HMI tags "2915RS001A01T01"
   "2915RS001A01T01.MSW" : 52809b66-421d-457f-8884-6f7a49d4e247 AT %DB5041.DBX18.0, 500 ms
   "2915RS001A01T01.DefaultText" : TextRef, internal   // Заголовок POPUP окна. При експорте из ECS через скрипт заполняется автоматически, если теги копируются в ручную то требуется в ручную задатать свойство Start Value
   "2915RS001A01T01.BlockInfo" : Array [0..2] of Int AT %DB5041.DBX38.0, 500 ms
   "2915RS001A01T01.StatusWork" : Int AT %DB5041.DBW242, 500 ms
   "2915RS001A01T01.FP_PARAM.DampingTime" : Int AT %DB5041.DBW50, 500 ms
   "2915RS001A01T01.FP_PARAM.Force_Value" : Real AT %DB5041.DBD52, 500 ms
   "2915RS001A01T01.FP_PARAM.Scale_Min" : Real AT %DB5041.DBD56, 500 ms
   "2915RS001A01T01.FP_PARAM.Scale_Max" : Real AT %DB5041.DBD60, 500 ms
   "2915RS001A01T01.FP_PARAM.Gradient" : Real AT %DB5041.DBD64, 500 ms
   "2915RS001A01T01.FP_PARAM.Grad_Pos" : Real AT %DB5041.DBD68, 500 ms
   "2915RS001A01T01.FP_PARAM.Grad_Neg" : Real AT %DB5041.DBD72, 500 ms
   "2915RS001A01T01.FP_PARAM.Grad_X" : Real AT %DB5041.DBD76, 500 ms
   "2915RS001A01T01.FP_PARAM.Gradient_Time_Pre" : Int AT %DB5041.DBW80, 500 ms
   "2915RS001A01T01.FP_PARAM.Gradient_Time_ACC" : Int AT %DB5041.DBW82, 500 ms
   "2915RS001A01T01.FP_PARAM.Alarm_Hyst" : Real AT %DB5041.DBD84, 500 ms
   "2915RS001A01T01.FP_PARAM.AlarmLimit_H3" : Real AT %DB5041.DBD88, 500 ms
   "2915RS001A01T01.FP_PARAM.AlarmLimit_H2" : Real AT %DB5041.DBD92, 500 ms
   "2915RS001A01T01.FP_PARAM.AlarmLimit_H1" : Real AT %DB5041.DBD96, 500 ms
   "2915RS001A01T01.FP_PARAM.AlarmLimit_L1" : Real AT %DB5041.DBD100, 500 ms
   "2915RS001A01T01.FP_PARAM.AlarmLimit_L2" : Real AT %DB5041.DBD104, 500 ms
   "2915RS001A01T01.FP_PARAM.AlarmLimit_L3" : Real AT %DB5041.DBD108, 500 ms
   "2915RS001A01T01.FP_PARAM.AlarmDelay_H3_Pre" : Int AT %DB5041.DBW112, 500 ms
   "2915RS001A01T01.FP_PARAM.AlarmDelay_H3_Acc" : Int AT %DB5041.DBW114, 500 ms
   "2915RS001A01T01.FP_PARAM.AlarmDelay_H2_Pre" : Int AT %DB5041.DBW116, 500 ms
   "2915RS001A01T01.FP_PARAM.AlarmDelay_H2_Acc" : Int AT %DB5041.DBW118, 500 ms
   "2915RS001A01T01.FP_PARAM.AlarmDelay_H1_Pre" : Int AT %DB5041.DBW120, 500 ms
   "2915RS001A01T01.FP_PARAM.AlarmDelay_H1_Acc" : Int AT %DB5041.DBW122, 500 ms
   "2915RS001A01T01.FP_PARAM.AlarmDelay_L1_Pre" : Int AT %DB5041.DBW124, 500 ms
   "2915RS001A01T01.FP_PARAM.AlarmDelay_L1_Acc" : Int AT %DB5041.DBW126, 500 ms
   "2915RS001A01T01.FP_PARAM.AlarmDelay_L2_Pre" : Int AT %DB5041.DBW128, 500 ms
   "2915RS001A01T01.FP_PARAM.AlarmDelay_L2_Acc" : Int AT %DB5041.DBW130, 500 ms
   "2915RS001A01T01.FP_PARAM.AlarmDelay_L3_Pre" : Int AT %DB5041.DBW132, 500 ms
   "2915RS001A01T01.FP_PARAM.AlarmDelay_L3_Acc" : Int AT %DB5041.DBW134, 500 ms
   "2915RS001A01T01.FP_PARAM.OpenLoopDelay_Pre" : Int AT %DB5041.DBW136, 500 ms
   "2915RS001A01T01.FP_PARAM.OpenLoopDelay_Acc" : Int AT %DB5041.DBW138, 500 ms
   "2915RS001A01T01.FP_PARAM.OverRangeDelay_Pre" : Int AT %DB5041.DBW140, 500 ms
   "2915RS001A01T01.FP_PARAM.OverRangeDelay_Acc" : Int AT %DB5041.DBW142, 500 ms
   "2915RS001A01T01.FP_PARAM.AuxLimit_H2_Value" : Real AT %DB5041.DBD144, 500 ms
   "2915RS001A01T01.FP_PARAM.AuxLimit_H1_Value" : Real AT %DB5041.DBD148, 500 ms
   "2915RS001A01T01.FP_PARAM.AuxLimit_L2_Value" : Real AT %DB5041.DBD152, 500 ms
   "2915RS001A01T01.FP_PARAM.AuxLimit_L1_Value" : Real AT %DB5041.DBD156, 500 ms
   "2915RS001A01T01.Unit" : TextRef, internal   // Еденицы измерения При експорте из ECS через скрипт заполняется автоматически, если теги копируются в ручную то требуется задатать свойство Text
   "2915RS001A01T01.Decimals" : TextRef, internal   // Формат отображения При експорте из ECS через скрипт, заполняется автоматически. Если теги копируются в ручную то требуется задатать свойство Text s999999.9
   "2915RS001A01T01.FP_EN.Square" : Bool AT %DB5041.DBX46.0, 500 ms
   "2915RS001A01T01.FP_EN.SquareRoot" : Bool AT %DB5041.DBX46.1, 500 ms
   "2915RS001A01T01.FP_EN.ParentSupress" : Bool AT %DB5041.DBX46.2, 500 ms
   "2915RS001A01T01.FP_EN.ParentSupressUnit" : Bool AT %DB5041.DBX46.3, 500 ms
   "2915RS001A01T01.FP_EN.Force" : Bool AT %DB5041.DBX46.4, 500 ms
   "2915RS001A01T01.FP_EN.Damping" : Bool AT %DB5041.DBX46.5, 500 ms
   "2915RS001A01T01.FP_EN.Gradient_Pos" : Bool AT %DB5041.DBX46.6, 500 ms
   "2915RS001A01T01.FP_EN.Gradient_Neg" : Bool AT %DB5041.DBX46.7, 500 ms
   "2915RS001A01T01.FP_EN.Hysteresis" : Bool AT %DB5041.DBX47.0, 500 ms
   "2915RS001A01T01.FP_EN.Alarm_H3" : Bool AT %DB5041.DBX47.1, 500 ms
   "2915RS001A01T01.FP_EN.Alarm_H2" : Bool AT %DB5041.DBX47.2, 500 ms
   "2915RS001A01T01.FP_EN.Alarm_H1" : Bool AT %DB5041.DBX47.3, 500 ms
   "2915RS001A01T01.FP_EN.Alarm_L1" : Bool AT %DB5041.DBX47.4, 500 ms
   "2915RS001A01T01.FP_EN.Alarm_L2" : Bool AT %DB5041.DBX47.5, 500 ms
   "2915RS001A01T01.FP_EN.Alarm_L3" : Bool AT %DB5041.DBX47.6, 500 ms
   "2915RS001A01T01.FP_EN.AlarmDelay_H3" : Bool AT %DB5041.DBX47.7, 500 ms
   "2915RS001A01T01.FP_EN.AlarmDelay_H2" : Bool AT %DB5041.DBX48.0, 500 ms
   "2915RS001A01T01.FP_EN.AlarmDelay_H1" : Bool AT %DB5041.DBX48.1, 500 ms
   "2915RS001A01T01.FP_EN.AlarmDelay_L1" : Bool AT %DB5041.DBX48.2, 500 ms
   "2915RS001A01T01.FP_EN.AlarmDelay_L2" : Bool AT %DB5041.DBX48.3, 500 ms
   "2915RS001A01T01.FP_EN.AlarmDelay_L3" : Bool AT %DB5041.DBX48.4, 500 ms
   "2915RS001A01T01.FP_EN.ROC_Warn" : Bool AT %DB5041.DBX48.5, 500 ms
   "2915RS001A01T01.FP_EN.U_Range_Warn" : Bool AT %DB5041.DBX48.6, 500 ms
   "2915RS001A01T01.FP_EN.O_Range_Warn" : Bool AT %DB5041.DBX48.7, 500 ms
   "2915RS001A01T01.trend_tag_name" : TextRef, internal   // Еденицы измерения При експорте из ECS через скрипт - заполняется автоматически, если теги копируются в ручную то требуется задатать свойство Text - имя тега для тренда
   "2915RS001A01T01.DQ.AL_H3" : Bool AT %DB5041.DBX16.0, 500 ms
   "2915RS001A01T01.DQ.AL_H2" : Bool AT %DB5041.DBX16.1, 500 ms
   "2915RS001A01T01.DQ.AL_H1" : Bool AT %DB5041.DBX16.2, 500 ms
   "2915RS001A01T01.DQ.AL_L1" : Bool AT %DB5041.DBX16.3, 500 ms
   "2915RS001A01T01.DQ.AL_L2" : Bool AT %DB5041.DBX16.4, 500 ms
   "2915RS001A01T01.DQ.AL_L3" : Bool AT %DB5041.DBX16.5, 500 ms
   "2915RS001A01T01.DQ.SIG_OK" : Bool AT %DB5041.DBX16.6, 500 ms
   "2915RS001A01T01.DQ.LIM_H2" : Bool AT %DB5041.DBX16.7, 500 ms
   "2915RS001A01T01.DQ.LIM_H1" : Bool AT %DB5041.DBX17.0, 500 ms
   "2915RS001A01T01.DQ.LIM_L1" : Bool AT %DB5041.DBX17.1, 500 ms
   "2915RS001A01T01.DQ.LIM_L2" : Bool AT %DB5041.DBX17.2, 500 ms
   "2915RS001A01T01.DQ.GR_P" : Bool AT %DB5041.DBX17.3, 500 ms
   "2915RS001A01T01.DQ.GR_N" : Bool AT %DB5041.DBX17.4, 500 ms
   "2915RS001A01T01.I.IN" : Real AT %DB5041.DBD2, 500 ms
   "2915RS001A01T01.I.SIG_TYPE" : Int AT %DB5041.DBW0, 500 ms
   "2915RS001A01T01.I.FI_BUS" : Byte AT %DB5041.DBB6, 500 ms
   "2915RS001A01T01.DI.U_RANGE" : Bool AT %DB5041.DBX7.0, 500 ms
   "2915RS001A01T01.DI.O_RANGE" : Bool AT %DB5041.DBX7.1, 500 ms
   "2915RS001A01T01.DI.SIG_FAULT" : Bool AT %DB5041.DBX7.2, 500 ms
   "2915RS001A01T01.DI.EnConfig" : Bool AT %DB5041.DBX7.3, 500 ms
   "2915RS001A01T01.DI.AEN" : Bool AT %DB5041.DBX7.4, 500 ms
   "2915RS001A01T01.DI.AL_SUPR" : Bool AT %DB5041.DBX7.5, 500 ms
   "2915RS001A01T01.Q.PV_NORM" : Real AT %DB5041.DBD8, 500 ms
   "2915RS001A01T01.Q.PV_SCAL" : Real AT %DB5041.DBD12, 500 ms
   "2915RS001A01T01.ParentInfo" : TextRef, internal   // Имя родителя для попап окна, вкладка инфо. При експорте из ECS через скрипт заполняется автоматически, если теги копируются в ручную то требуется в ручную задатать свойство Start Value

HMI tags "2915RS001A01T02"
   "2915RS001A01T02.MSW" : 52809b66-421d-457f-8884-6f7a49d4e247 AT %DB5042.DBX18.0, 500 ms
   "2915RS001A01T02.DefaultText" : TextRef, internal   // Заголовок POPUP окна. При експорте из ECS через скрипт заполняется автоматически, если теги копируются в ручную то требуется в ручную задатать свойство Start Value
   "2915RS001A01T02.BlockInfo" : Array [0..2] of Int AT %DB5042.DBX38.0, 500 ms
   "2915RS001A01T02.StatusWork" : Int AT %DB5042.DBW242, 500 ms
   "2915RS001A01T02.FP_PARAM.DampingTime" : Int AT %DB5042.DBW50, 500 ms
   "2915RS001A01T02.FP_PARAM.Force_Value" : Real AT %DB5042.DBD52, 500 ms
   "2915RS001A01T02.FP_PARAM.Scale_Min" : Real AT %DB5042.DBD56, 500 ms
   "2915RS001A01T02.FP_PARAM.Scale_Max" : Real AT %DB5042.DBD60, 500 ms
   "2915RS001A01T02.FP_PARAM.Gradient" : Real AT %DB5042.DBD64, 500 ms
   "2915RS001A01T02.FP_PARAM.Grad_Pos" : Real AT %DB5042.DBD68, 500 ms
   "2915RS001A01T02.FP_PARAM.Grad_Neg" : Real AT %DB5042.DBD72, 500 ms
   "2915RS001A01T02.FP_PARAM.Grad_X" : Real AT %DB5042.DBD76, 500 ms
   "2915RS001A01T02.FP_PARAM.Gradient_Time_Pre" : Int AT %DB5042.DBW80, 500 ms
   "2915RS001A01T02.FP_PARAM.Gradient_Time_ACC" : Int AT %DB5042.DBW82, 500 ms
   "2915RS001A01T02.FP_PARAM.Alarm_Hyst" : Real AT %DB5042.DBD84, 500 ms
   "2915RS001A01T02.FP_PARAM.AlarmLimit_H3" : Real AT %DB5042.DBD88, 500 ms
   "2915RS001A01T02.FP_PARAM.AlarmLimit_H2" : Real AT %DB5042.DBD92, 500 ms
   "2915RS001A01T02.FP_PARAM.AlarmLimit_H1" : Real AT %DB5042.DBD96, 500 ms
   "2915RS001A01T02.FP_PARAM.AlarmLimit_L1" : Real AT %DB5042.DBD100, 500 ms
   "2915RS001A01T02.FP_PARAM.AlarmLimit_L2" : Real AT %DB5042.DBD104, 500 ms
   "2915RS001A01T02.FP_PARAM.AlarmLimit_L3" : Real AT %DB5042.DBD108, 500 ms
   "2915RS001A01T02.FP_PARAM.AlarmDelay_H3_Pre" : Int AT %DB5042.DBW112, 500 ms
   "2915RS001A01T02.FP_PARAM.AlarmDelay_H3_Acc" : Int AT %DB5042.DBW114, 500 ms
   "2915RS001A01T02.FP_PARAM.AlarmDelay_H2_Pre" : Int AT %DB5042.DBW116, 500 ms
   "2915RS001A01T02.FP_PARAM.AlarmDelay_H2_Acc" : Int AT %DB5042.DBW118, 500 ms
   "2915RS001A01T02.FP_PARAM.AlarmDelay_H1_Pre" : Int AT %DB5042.DBW120, 500 ms
   "2915RS001A01T02.FP_PARAM.AlarmDelay_H1_Acc" : Int AT %DB5042.DBW122, 500 ms
   "2915RS001A01T02.FP_PARAM.AlarmDelay_L1_Pre" : Int AT %DB5042.DBW124, 500 ms
   "2915RS001A01T02.FP_PARAM.AlarmDelay_L1_Acc" : Int AT %DB5042.DBW126, 500 ms
   "2915RS001A01T02.FP_PARAM.AlarmDelay_L2_Pre" : Int AT %DB5042.DBW128, 500 ms
   "2915RS001A01T02.FP_PARAM.AlarmDelay_L2_Acc" : Int AT %DB5042.DBW130, 500 ms
   "2915RS001A01T02.FP_PARAM.AlarmDelay_L3_Pre" : Int AT %DB5042.DBW132, 500 ms
   "2915RS001A01T02.FP_PARAM.AlarmDelay_L3_Acc" : Int AT %DB5042.DBW134, 500 ms
   "2915RS001A01T02.FP_PARAM.OpenLoopDelay_Pre" : Int AT %DB5042.DBW136, 500 ms
   "2915RS001A01T02.FP_PARAM.OpenLoopDelay_Acc" : Int AT %DB5042.DBW138, 500 ms
   "2915RS001A01T02.FP_PARAM.OverRangeDelay_Pre" : Int AT %DB5042.DBW140, 500 ms
   "2915RS001A01T02.FP_PARAM.OverRangeDelay_Acc" : Int AT %DB5042.DBW142, 500 ms
   "2915RS001A01T02.FP_PARAM.AuxLimit_H2_Value" : Real AT %DB5042.DBD144, 500 ms
   "2915RS001A01T02.FP_PARAM.AuxLimit_H1_Value" : Real AT %DB5042.DBD148, 500 ms
   "2915RS001A01T02.FP_PARAM.AuxLimit_L2_Value" : Real AT %DB5042.DBD152, 500 ms
   "2915RS001A01T02.FP_PARAM.AuxLimit_L1_Value" : Real AT %DB5042.DBD156, 500 ms
   "2915RS001A01T02.Unit" : TextRef, internal   // Еденицы измерения При експорте из ECS через скрипт заполняется автоматически, если теги копируются в ручную то требуется задатать свойство Text
   "2915RS001A01T02.Decimals" : TextRef, internal   // Формат отображения При експорте из ECS через скрипт, заполняется автоматически. Если теги копируются в ручную то требуется задатать свойство Text s999999.9
   "2915RS001A01T02.FP_EN.Square" : Bool AT %DB5042.DBX46.0, 500 ms
   "2915RS001A01T02.FP_EN.SquareRoot" : Bool AT %DB5042.DBX46.1, 500 ms
   "2915RS001A01T02.FP_EN.ParentSupress" : Bool AT %DB5042.DBX46.2, 500 ms
   "2915RS001A01T02.FP_EN.ParentSupressUnit" : Bool AT %DB5042.DBX46.3, 500 ms
   "2915RS001A01T02.FP_EN.Force" : Bool AT %DB5042.DBX46.4, 500 ms
   "2915RS001A01T02.FP_EN.Damping" : Bool AT %DB5042.DBX46.5, 500 ms
   "2915RS001A01T02.FP_EN.Gradient_Pos" : Bool AT %DB5042.DBX46.6, 500 ms
   "2915RS001A01T02.FP_EN.Gradient_Neg" : Bool AT %DB5042.DBX46.7, 500 ms
   "2915RS001A01T02.FP_EN.Hysteresis" : Bool AT %DB5042.DBX47.0, 500 ms
   "2915RS001A01T02.FP_EN.Alarm_H3" : Bool AT %DB5042.DBX47.1, 500 ms
   "2915RS001A01T02.FP_EN.Alarm_H2" : Bool AT %DB5042.DBX47.2, 500 ms
   "2915RS001A01T02.FP_EN.Alarm_H1" : Bool AT %DB5042.DBX47.3, 500 ms
   "2915RS001A01T02.FP_EN.Alarm_L1" : Bool AT %DB5042.DBX47.4, 500 ms
   "2915RS001A01T02.FP_EN.Alarm_L2" : Bool AT %DB5042.DBX47.5, 500 ms
   "2915RS001A01T02.FP_EN.Alarm_L3" : Bool AT %DB5042.DBX47.6, 500 ms
   "2915RS001A01T02.FP_EN.AlarmDelay_H3" : Bool AT %DB5042.DBX47.7, 500 ms
   "2915RS001A01T02.FP_EN.AlarmDelay_H2" : Bool AT %DB5042.DBX48.0, 500 ms
   "2915RS001A01T02.FP_EN.AlarmDelay_H1" : Bool AT %DB5042.DBX48.1, 500 ms
   "2915RS001A01T02.FP_EN.AlarmDelay_L1" : Bool AT %DB5042.DBX48.2, 500 ms
   "2915RS001A01T02.FP_EN.AlarmDelay_L2" : Bool AT %DB5042.DBX48.3, 500 ms
   "2915RS001A01T02.FP_EN.AlarmDelay_L3" : Bool AT %DB5042.DBX48.4, 500 ms
   "2915RS001A01T02.FP_EN.ROC_Warn" : Bool AT %DB5042.DBX48.5, 500 ms
   "2915RS001A01T02.FP_EN.U_Range_Warn" : Bool AT %DB5042.DBX48.6, 500 ms
   "2915RS001A01T02.FP_EN.O_Range_Warn" : Bool AT %DB5042.DBX48.7, 500 ms
   "2915RS001A01T02.trend_tag_name" : TextRef, internal   // Еденицы измерения При експорте из ECS через скрипт - заполняется автоматически, если теги копируются в ручную то требуется задатать свойство Text - имя тега для тренда
   "2915RS001A01T02.DQ.AL_H3" : Bool AT %DB5042.DBX16.0, 500 ms
   "2915RS001A01T02.DQ.AL_H2" : Bool AT %DB5042.DBX16.1, 500 ms
   "2915RS001A01T02.DQ.AL_H1" : Bool AT %DB5042.DBX16.2, 500 ms
   "2915RS001A01T02.DQ.AL_L1" : Bool AT %DB5042.DBX16.3, 500 ms
   "2915RS001A01T02.DQ.AL_L2" : Bool AT %DB5042.DBX16.4, 500 ms
   "2915RS001A01T02.DQ.AL_L3" : Bool AT %DB5042.DBX16.5, 500 ms
   "2915RS001A01T02.DQ.SIG_OK" : Bool AT %DB5042.DBX16.6, 500 ms
   "2915RS001A01T02.DQ.LIM_H2" : Bool AT %DB5042.DBX16.7, 500 ms
   "2915RS001A01T02.DQ.LIM_H1" : Bool AT %DB5042.DBX17.0, 500 ms
   "2915RS001A01T02.DQ.LIM_L1" : Bool AT %DB5042.DBX17.1, 500 ms
   "2915RS001A01T02.DQ.LIM_L2" : Bool AT %DB5042.DBX17.2, 500 ms
   "2915RS001A01T02.DQ.GR_P" : Bool AT %DB5042.DBX17.3, 500 ms
   "2915RS001A01T02.DQ.GR_N" : Bool AT %DB5042.DBX17.4, 500 ms
   "2915RS001A01T02.I.IN" : Real AT %DB5042.DBD2, 500 ms
   "2915RS001A01T02.I.SIG_TYPE" : Int AT %DB5042.DBW0, 500 ms
   "2915RS001A01T02.I.FI_BUS" : Byte AT %DB5042.DBB6, 500 ms
   "2915RS001A01T02.DI.U_RANGE" : Bool AT %DB5042.DBX7.0, 500 ms
   "2915RS001A01T02.DI.O_RANGE" : Bool AT %DB5042.DBX7.1, 500 ms
   "2915RS001A01T02.DI.SIG_FAULT" : Bool AT %DB5042.DBX7.2, 500 ms
   "2915RS001A01T02.DI.EnConfig" : Bool AT %DB5042.DBX7.3, 500 ms
   "2915RS001A01T02.DI.AEN" : Bool AT %DB5042.DBX7.4, 500 ms
   "2915RS001A01T02.DI.AL_SUPR" : Bool AT %DB5042.DBX7.5, 500 ms
   "2915RS001A01T02.Q.PV_NORM" : Real AT %DB5042.DBD8, 500 ms
   "2915RS001A01T02.Q.PV_SCAL" : Real AT %DB5042.DBD12, 500 ms
   "2915RS001A01T02.ParentInfo" : TextRef, internal   // Имя родителя для попап окна, вкладка инфо. При експорте из ECS через скрипт заполняется автоматически, если теги копируются в ручную то требуется в ручную задатать свойство Start Value

HMI tags "2915RS001A01T03"
   "2915RS001A01T03.MSW" : 52809b66-421d-457f-8884-6f7a49d4e247 AT %DB5043.DBX18.0, 500 ms
   "2915RS001A01T03.DefaultText" : TextRef, internal   // Заголовок POPUP окна. При експорте из ECS через скрипт заполняется автоматически, если теги копируются в ручную то требуется в ручную задатать свойство Start Value
   "2915RS001A01T03.BlockInfo" : Array [0..2] of Int AT %DB5043.DBX38.0, 500 ms
   "2915RS001A01T03.StatusWork" : Int AT %DB5043.DBW242, 500 ms
   "2915RS001A01T03.FP_PARAM.DampingTime" : Int AT %DB5043.DBW50, 500 ms
   "2915RS001A01T03.FP_PARAM.Force_Value" : Real AT %DB5043.DBD52, 500 ms
   "2915RS001A01T03.FP_PARAM.Scale_Min" : Real AT %DB5043.DBD56, 500 ms
   "2915RS001A01T03.FP_PARAM.Scale_Max" : Real AT %DB5043.DBD60, 500 ms
   "2915RS001A01T03.FP_PARAM.Gradient" : Real AT %DB5043.DBD64, 500 ms
   "2915RS001A01T03.FP_PARAM.Grad_Pos" : Real AT %DB5043.DBD68, 500 ms
   "2915RS001A01T03.FP_PARAM.Grad_Neg" : Real AT %DB5043.DBD72, 500 ms
   "2915RS001A01T03.FP_PARAM.Grad_X" : Real AT %DB5043.DBD76, 500 ms
   "2915RS001A01T03.FP_PARAM.Gradient_Time_Pre" : Int AT %DB5043.DBW80, 500 ms
   "2915RS001A01T03.FP_PARAM.Gradient_Time_ACC" : Int AT %DB5043.DBW82, 500 ms
   "2915RS001A01T03.FP_PARAM.Alarm_Hyst" : Real AT %DB5043.DBD84, 500 ms
   "2915RS001A01T03.FP_PARAM.AlarmLimit_H3" : Real AT %DB5043.DBD88, 500 ms
   "2915RS001A01T03.FP_PARAM.AlarmLimit_H2" : Real AT %DB5043.DBD92, 500 ms
   "2915RS001A01T03.FP_PARAM.AlarmLimit_H1" : Real AT %DB5043.DBD96, 500 ms
   "2915RS001A01T03.FP_PARAM.AlarmLimit_L1" : Real AT %DB5043.DBD100, 500 ms
   "2915RS001A01T03.FP_PARAM.AlarmLimit_L2" : Real AT %DB5043.DBD104, 500 ms
   "2915RS001A01T03.FP_PARAM.AlarmLimit_L3" : Real AT %DB5043.DBD108, 500 ms
   "2915RS001A01T03.FP_PARAM.AlarmDelay_H3_Pre" : Int AT %DB5043.DBW112, 500 ms
   "2915RS001A01T03.FP_PARAM.AlarmDelay_H3_Acc" : Int AT %DB5043.DBW114, 500 ms
   "2915RS001A01T03.FP_PARAM.AlarmDelay_H2_Pre" : Int AT %DB5043.DBW116, 500 ms
   "2915RS001A01T03.FP_PARAM.AlarmDelay_H2_Acc" : Int AT %DB5043.DBW118, 500 ms
   "2915RS001A01T03.FP_PARAM.AlarmDelay_H1_Pre" : Int AT %DB5043.DBW120, 500 ms
   "2915RS001A01T03.FP_PARAM.AlarmDelay_H1_Acc" : Int AT %DB5043.DBW122, 500 ms
   "2915RS001A01T03.FP_PARAM.AlarmDelay_L1_Pre" : Int AT %DB5043.DBW124, 500 ms
   "2915RS001A01T03.FP_PARAM.AlarmDelay_L1_Acc" : Int AT %DB5043.DBW126, 500 ms
   "2915RS001A01T03.FP_PARAM.AlarmDelay_L2_Pre" : Int AT %DB5043.DBW128, 500 ms
   "2915RS001A01T03.FP_PARAM.AlarmDelay_L2_Acc" : Int AT %DB5043.DBW130, 500 ms
   "2915RS001A01T03.FP_PARAM.AlarmDelay_L3_Pre" : Int AT %DB5043.DBW132, 500 ms
   "2915RS001A01T03.FP_PARAM.AlarmDelay_L3_Acc" : Int AT %DB5043.DBW134, 500 ms
   "2915RS001A01T03.FP_PARAM.OpenLoopDelay_Pre" : Int AT %DB5043.DBW136, 500 ms
   "2915RS001A01T03.FP_PARAM.OpenLoopDelay_Acc" : Int AT %DB5043.DBW138, 500 ms
   "2915RS001A01T03.FP_PARAM.OverRangeDelay_Pre" : Int AT %DB5043.DBW140, 500 ms
   "2915RS001A01T03.FP_PARAM.OverRangeDelay_Acc" : Int AT %DB5043.DBW142, 500 ms
   "2915RS001A01T03.FP_PARAM.AuxLimit_H2_Value" : Real AT %DB5043.DBD144, 500 ms
   "2915RS001A01T03.FP_PARAM.AuxLimit_H1_Value" : Real AT %DB5043.DBD148, 500 ms
   "2915RS001A01T03.FP_PARAM.AuxLimit_L2_Value" : Real AT %DB5043.DBD152, 500 ms
   "2915RS001A01T03.FP_PARAM.AuxLimit_L1_Value" : Real AT %DB5043.DBD156, 500 ms
   "2915RS001A01T03.Unit" : TextRef, internal   // Еденицы измерения При експорте из ECS через скрипт заполняется автоматически, если теги копируются в ручную то требуется задатать свойство Text
   "2915RS001A01T03.Decimals" : TextRef, internal   // Формат отображения При експорте из ECS через скрипт, заполняется автоматически. Если теги копируются в ручную то требуется задатать свойство Text s999999.9
   "2915RS001A01T03.FP_EN.Square" : Bool AT %DB5043.DBX46.0, 500 ms
   "2915RS001A01T03.FP_EN.SquareRoot" : Bool AT %DB5043.DBX46.1, 500 ms
   "2915RS001A01T03.FP_EN.ParentSupress" : Bool AT %DB5043.DBX46.2, 500 ms
   "2915RS001A01T03.FP_EN.ParentSupressUnit" : Bool AT %DB5043.DBX46.3, 500 ms
   "2915RS001A01T03.FP_EN.Force" : Bool AT %DB5043.DBX46.4, 500 ms
   "2915RS001A01T03.FP_EN.Damping" : Bool AT %DB5043.DBX46.5, 500 ms
   "2915RS001A01T03.FP_EN.Gradient_Pos" : Bool AT %DB5043.DBX46.6, 500 ms
   "2915RS001A01T03.FP_EN.Gradient_Neg" : Bool AT %DB5043.DBX46.7, 500 ms
   "2915RS001A01T03.FP_EN.Hysteresis" : Bool AT %DB5043.DBX47.0, 500 ms
   "2915RS001A01T03.FP_EN.Alarm_H3" : Bool AT %DB5043.DBX47.1, 500 ms
   "2915RS001A01T03.FP_EN.Alarm_H2" : Bool AT %DB5043.DBX47.2, 500 ms
   "2915RS001A01T03.FP_EN.Alarm_H1" : Bool AT %DB5043.DBX47.3, 500 ms
   "2915RS001A01T03.FP_EN.Alarm_L1" : Bool AT %DB5043.DBX47.4, 500 ms
   "2915RS001A01T03.FP_EN.Alarm_L2" : Bool AT %DB5043.DBX47.5, 500 ms
   "2915RS001A01T03.FP_EN.Alarm_L3" : Bool AT %DB5043.DBX47.6, 500 ms
   "2915RS001A01T03.FP_EN.AlarmDelay_H3" : Bool AT %DB5043.DBX47.7, 500 ms
   "2915RS001A01T03.FP_EN.AlarmDelay_H2" : Bool AT %DB5043.DBX48.0, 500 ms
   "2915RS001A01T03.FP_EN.AlarmDelay_H1" : Bool AT %DB5043.DBX48.1, 500 ms
   "2915RS001A01T03.FP_EN.AlarmDelay_L1" : Bool AT %DB5043.DBX48.2, 500 ms
   "2915RS001A01T03.FP_EN.AlarmDelay_L2" : Bool AT %DB5043.DBX48.3, 500 ms
   "2915RS001A01T03.FP_EN.AlarmDelay_L3" : Bool AT %DB5043.DBX48.4, 500 ms
   "2915RS001A01T03.FP_EN.ROC_Warn" : Bool AT %DB5043.DBX48.5, 500 ms
   "2915RS001A01T03.FP_EN.U_Range_Warn" : Bool AT %DB5043.DBX48.6, 500 ms
   "2915RS001A01T03.FP_EN.O_Range_Warn" : Bool AT %DB5043.DBX48.7, 500 ms
   "2915RS001A01T03.trend_tag_name" : TextRef, internal   // Еденицы измерения При експорте из ECS через скрипт - заполняется автоматически, если теги копируются в ручную то требуется задатать свойство Text - имя тега для тренда
   "2915RS001A01T03.DQ.AL_H3" : Bool AT %DB5043.DBX16.0, 500 ms
   "2915RS001A01T03.DQ.AL_H2" : Bool AT %DB5043.DBX16.1, 500 ms
   "2915RS001A01T03.DQ.AL_H1" : Bool AT %DB5043.DBX16.2, 500 ms
   "2915RS001A01T03.DQ.AL_L1" : Bool AT %DB5043.DBX16.3, 500 ms
   "2915RS001A01T03.DQ.AL_L2" : Bool AT %DB5043.DBX16.4, 500 ms
   "2915RS001A01T03.DQ.AL_L3" : Bool AT %DB5043.DBX16.5, 500 ms
   "2915RS001A01T03.DQ.SIG_OK" : Bool AT %DB5043.DBX16.6, 500 ms
   "2915RS001A01T03.DQ.LIM_H2" : Bool AT %DB5043.DBX16.7, 500 ms
   "2915RS001A01T03.DQ.LIM_H1" : Bool AT %DB5043.DBX17.0, 500 ms
   "2915RS001A01T03.DQ.LIM_L1" : Bool AT %DB5043.DBX17.1, 500 ms
   "2915RS001A01T03.DQ.LIM_L2" : Bool AT %DB5043.DBX17.2, 500 ms
   "2915RS001A01T03.DQ.GR_P" : Bool AT %DB5043.DBX17.3, 500 ms
   "2915RS001A01T03.DQ.GR_N" : Bool AT %DB5043.DBX17.4, 500 ms
   "2915RS001A01T03.I.IN" : Real AT %DB5043.DBD2, 500 ms
   "2915RS001A01T03.I.SIG_TYPE" : Int AT %DB5043.DBW0, 500 ms
   "2915RS001A01T03.I.FI_BUS" : Byte AT %DB5043.DBB6, 500 ms
   "2915RS001A01T03.DI.U_RANGE" : Bool AT %DB5043.DBX7.0, 500 ms
   "2915RS001A01T03.DI.O_RANGE" : Bool AT %DB5043.DBX7.1, 500 ms
   "2915RS001A01T03.DI.SIG_FAULT" : Bool AT %DB5043.DBX7.2, 500 ms
   "2915RS001A01T03.DI.EnConfig" : Bool AT %DB5043.DBX7.3, 500 ms
   "2915RS001A01T03.DI.AEN" : Bool AT %DB5043.DBX7.4, 500 ms
   "2915RS001A01T03.DI.AL_SUPR" : Bool AT %DB5043.DBX7.5, 500 ms
   "2915RS001A01T03.Q.PV_NORM" : Real AT %DB5043.DBD8, 500 ms
   "2915RS001A01T03.Q.PV_SCAL" : Real AT %DB5043.DBD12, 500 ms
   "2915RS001A01T03.ParentInfo" : TextRef, internal   // Имя родителя для попап окна, вкладка инфо. При експорте из ECS через скрипт заполняется автоматически, если теги копируются в ручную то требуется в ручную задатать свойство Start Value

HMI tags "2915RS001A01T04"
   "2915RS001A01T04.MSW" : 52809b66-421d-457f-8884-6f7a49d4e247 AT %DB5044.DBX18.0, 500 ms
   "2915RS001A01T04.DefaultText" : TextRef, internal   // Заголовок POPUP окна. При експорте из ECS через скрипт заполняется автоматически, если теги копируются в ручную то требуется в ручную задатать свойство Start Value
   "2915RS001A01T04.BlockInfo" : Array [0..2] of Int AT %DB5044.DBX38.0, 500 ms
   "2915RS001A01T04.StatusWork" : Int AT %DB5044.DBW242, 500 ms
   "2915RS001A01T04.FP_PARAM.DampingTime" : Int AT %DB5044.DBW50, 500 ms
   "2915RS001A01T04.FP_PARAM.Force_Value" : Real AT %DB5044.DBD52, 500 ms
   "2915RS001A01T04.FP_PARAM.Scale_Min" : Real AT %DB5044.DBD56, 500 ms
   "2915RS001A01T04.FP_PARAM.Scale_Max" : Real AT %DB5044.DBD60, 500 ms
   "2915RS001A01T04.FP_PARAM.Gradient" : Real AT %DB5044.DBD64, 500 ms
   "2915RS001A01T04.FP_PARAM.Grad_Pos" : Real AT %DB5044.DBD68, 500 ms
   "2915RS001A01T04.FP_PARAM.Grad_Neg" : Real AT %DB5044.DBD72, 500 ms
   "2915RS001A01T04.FP_PARAM.Grad_X" : Real AT %DB5044.DBD76, 500 ms
   "2915RS001A01T04.FP_PARAM.Gradient_Time_Pre" : Int AT %DB5044.DBW80, 500 ms
   "2915RS001A01T04.FP_PARAM.Gradient_Time_ACC" : Int AT %DB5044.DBW82, 500 ms
   "2915RS001A01T04.FP_PARAM.Alarm_Hyst" : Real AT %DB5044.DBD84, 500 ms
   "2915RS001A01T04.FP_PARAM.AlarmLimit_H3" : Real AT %DB5044.DBD88, 500 ms
   "2915RS001A01T04.FP_PARAM.AlarmLimit_H2" : Real AT %DB5044.DBD92, 500 ms
   "2915RS001A01T04.FP_PARAM.AlarmLimit_H1" : Real AT %DB5044.DBD96, 500 ms
   "2915RS001A01T04.FP_PARAM.AlarmLimit_L1" : Real AT %DB5044.DBD100, 500 ms
   "2915RS001A01T04.FP_PARAM.AlarmLimit_L2" : Real AT %DB5044.DBD104, 500 ms
   "2915RS001A01T04.FP_PARAM.AlarmLimit_L3" : Real AT %DB5044.DBD108, 500 ms
   "2915RS001A01T04.FP_PARAM.AlarmDelay_H3_Pre" : Int AT %DB5044.DBW112, 500 ms
   "2915RS001A01T04.FP_PARAM.AlarmDelay_H3_Acc" : Int AT %DB5044.DBW114, 500 ms
   "2915RS001A01T04.FP_PARAM.AlarmDelay_H2_Pre" : Int AT %DB5044.DBW116, 500 ms
   "2915RS001A01T04.FP_PARAM.AlarmDelay_H2_Acc" : Int AT %DB5044.DBW118, 500 ms
   "2915RS001A01T04.FP_PARAM.AlarmDelay_H1_Pre" : Int AT %DB5044.DBW120, 500 ms
   "2915RS001A01T04.FP_PARAM.AlarmDelay_H1_Acc" : Int AT %DB5044.DBW122, 500 ms
   "2915RS001A01T04.FP_PARAM.AlarmDelay_L1_Pre" : Int AT %DB5044.DBW124, 500 ms
   "2915RS001A01T04.FP_PARAM.AlarmDelay_L1_Acc" : Int AT %DB5044.DBW126, 500 ms
   "2915RS001A01T04.FP_PARAM.AlarmDelay_L2_Pre" : Int AT %DB5044.DBW128, 500 ms
   "2915RS001A01T04.FP_PARAM.AlarmDelay_L2_Acc" : Int AT %DB5044.DBW130, 500 ms
   "2915RS001A01T04.FP_PARAM.AlarmDelay_L3_Pre" : Int AT %DB5044.DBW132, 500 ms
   "2915RS001A01T04.FP_PARAM.AlarmDelay_L3_Acc" : Int AT %DB5044.DBW134, 500 ms
   "2915RS001A01T04.FP_PARAM.OpenLoopDelay_Pre" : Int AT %DB5044.DBW136, 500 ms
   "2915RS001A01T04.FP_PARAM.OpenLoopDelay_Acc" : Int AT %DB5044.DBW138, 500 ms
   "2915RS001A01T04.FP_PARAM.OverRangeDelay_Pre" : Int AT %DB5044.DBW140, 500 ms
   "2915RS001A01T04.FP_PARAM.OverRangeDelay_Acc" : Int AT %DB5044.DBW142, 500 ms
   "2915RS001A01T04.FP_PARAM.AuxLimit_H2_Value" : Real AT %DB5044.DBD144, 500 ms
   "2915RS001A01T04.FP_PARAM.AuxLimit_H1_Value" : Real AT %DB5044.DBD148, 500 ms
   "2915RS001A01T04.FP_PARAM.AuxLimit_L2_Value" : Real AT %DB5044.DBD152, 500 ms
   "2915RS001A01T04.FP_PARAM.AuxLimit_L1_Value" : Real AT %DB5044.DBD156, 500 ms
   "2915RS001A01T04.Unit" : TextRef, internal   // Еденицы измерения При експорте из ECS через скрипт заполняется автоматически, если теги копируются в ручную то требуется задатать свойство Text
   "2915RS001A01T04.Decimals" : TextRef, internal   // Формат отображения При експорте из ECS через скрипт, заполняется автоматически. Если теги копируются в ручную то требуется задатать свойство Text s999999.9
   "2915RS001A01T04.FP_EN.Square" : Bool AT %DB5044.DBX46.0, 500 ms
   "2915RS001A01T04.FP_EN.SquareRoot" : Bool AT %DB5044.DBX46.1, 500 ms
   "2915RS001A01T04.FP_EN.ParentSupress" : Bool AT %DB5044.DBX46.2, 500 ms
   "2915RS001A01T04.FP_EN.ParentSupressUnit" : Bool AT %DB5044.DBX46.3, 500 ms
   "2915RS001A01T04.FP_EN.Force" : Bool AT %DB5044.DBX46.4, 500 ms
   "2915RS001A01T04.FP_EN.Damping" : Bool AT %DB5044.DBX46.5, 500 ms
   "2915RS001A01T04.FP_EN.Gradient_Pos" : Bool AT %DB5044.DBX46.6, 500 ms
   "2915RS001A01T04.FP_EN.Gradient_Neg" : Bool AT %DB5044.DBX46.7, 500 ms
   "2915RS001A01T04.FP_EN.Hysteresis" : Bool AT %DB5044.DBX47.0, 500 ms
   "2915RS001A01T04.FP_EN.Alarm_H3" : Bool AT %DB5044.DBX47.1, 500 ms
   "2915RS001A01T04.FP_EN.Alarm_H2" : Bool AT %DB5044.DBX47.2, 500 ms
   "2915RS001A01T04.FP_EN.Alarm_H1" : Bool AT %DB5044.DBX47.3, 500 ms
   "2915RS001A01T04.FP_EN.Alarm_L1" : Bool AT %DB5044.DBX47.4, 500 ms
   "2915RS001A01T04.FP_EN.Alarm_L2" : Bool AT %DB5044.DBX47.5, 500 ms
   "2915RS001A01T04.FP_EN.Alarm_L3" : Bool AT %DB5044.DBX47.6, 500 ms
   "2915RS001A01T04.FP_EN.AlarmDelay_H3" : Bool AT %DB5044.DBX47.7, 500 ms
   "2915RS001A01T04.FP_EN.AlarmDelay_H2" : Bool AT %DB5044.DBX48.0, 500 ms
   "2915RS001A01T04.FP_EN.AlarmDelay_H1" : Bool AT %DB5044.DBX48.1, 500 ms
   "2915RS001A01T04.FP_EN.AlarmDelay_L1" : Bool AT %DB5044.DBX48.2, 500 ms
   "2915RS001A01T04.FP_EN.AlarmDelay_L2" : Bool AT %DB5044.DBX48.3, 500 ms
   "2915RS001A01T04.FP_EN.AlarmDelay_L3" : Bool AT %DB5044.DBX48.4, 500 ms
   "2915RS001A01T04.FP_EN.ROC_Warn" : Bool AT %DB5044.DBX48.5, 500 ms
   "2915RS001A01T04.FP_EN.U_Range_Warn" : Bool AT %DB5044.DBX48.6, 500 ms
   "2915RS001A01T04.FP_EN.O_Range_Warn" : Bool AT %DB5044.DBX48.7, 500 ms
   "2915RS001A01T04.trend_tag_name" : TextRef, internal   // Еденицы измерения При експорте из ECS через скрипт - заполняется автоматически, если теги копируются в ручную то требуется задатать свойство Text - имя тега для тренда
   "2915RS001A01T04.DQ.AL_H3" : Bool AT %DB5044.DBX16.0, 500 ms
   "2915RS001A01T04.DQ.AL_H2" : Bool AT %DB5044.DBX16.1, 500 ms
   "2915RS001A01T04.DQ.AL_H1" : Bool AT %DB5044.DBX16.2, 500 ms
   "2915RS001A01T04.DQ.AL_L1" : Bool AT %DB5044.DBX16.3, 500 ms
   "2915RS001A01T04.DQ.AL_L2" : Bool AT %DB5044.DBX16.4, 500 ms
   "2915RS001A01T04.DQ.AL_L3" : Bool AT %DB5044.DBX16.5, 500 ms
   "2915RS001A01T04.DQ.SIG_OK" : Bool AT %DB5044.DBX16.6, 500 ms
   "2915RS001A01T04.DQ.LIM_H2" : Bool AT %DB5044.DBX16.7, 500 ms
   "2915RS001A01T04.DQ.LIM_H1" : Bool AT %DB5044.DBX17.0, 500 ms
   "2915RS001A01T04.DQ.LIM_L1" : Bool AT %DB5044.DBX17.1, 500 ms
   "2915RS001A01T04.DQ.LIM_L2" : Bool AT %DB5044.DBX17.2, 500 ms
   "2915RS001A01T04.DQ.GR_P" : Bool AT %DB5044.DBX17.3, 500 ms
   "2915RS001A01T04.DQ.GR_N" : Bool AT %DB5044.DBX17.4, 500 ms
   "2915RS001A01T04.I.IN" : Real AT %DB5044.DBD2, 500 ms
   "2915RS001A01T04.I.SIG_TYPE" : Int AT %DB5044.DBW0, 500 ms
   "2915RS001A01T04.I.FI_BUS" : Byte AT %DB5044.DBB6, 500 ms
   "2915RS001A01T04.DI.U_RANGE" : Bool AT %DB5044.DBX7.0, 500 ms
   "2915RS001A01T04.DI.O_RANGE" : Bool AT %DB5044.DBX7.1, 500 ms
   "2915RS001A01T04.DI.SIG_FAULT" : Bool AT %DB5044.DBX7.2, 500 ms
   "2915RS001A01T04.DI.EnConfig" : Bool AT %DB5044.DBX7.3, 500 ms
   "2915RS001A01T04.DI.AEN" : Bool AT %DB5044.DBX7.4, 500 ms
   "2915RS001A01T04.DI.AL_SUPR" : Bool AT %DB5044.DBX7.5, 500 ms
   "2915RS001A01T04.Q.PV_NORM" : Real AT %DB5044.DBD8, 500 ms
   "2915RS001A01T04.Q.PV_SCAL" : Real AT %DB5044.DBD12, 500 ms
   "2915RS001A01T04.ParentInfo" : TextRef, internal   // Имя родителя для попап окна, вкладка инфо. При експорте из ECS через скрипт заполняется автоматически, если теги копируются в ручную то требуется в ручную задатать свойство Start Value

HMI tags "2915RS001A01T05"
   "2915RS001A01T05.MSW" : 52809b66-421d-457f-8884-6f7a49d4e247 AT %DB5045.DBX18.0, 500 ms
   "2915RS001A01T05.DefaultText" : TextRef, internal   // Заголовок POPUP окна. При експорте из ECS через скрипт заполняется автоматически, если теги копируются в ручную то требуется в ручную задатать свойство Start Value
   "2915RS001A01T05.BlockInfo" : Array [0..2] of Int AT %DB5045.DBX38.0, 500 ms
   "2915RS001A01T05.StatusWork" : Int AT %DB5045.DBW242, 500 ms
   "2915RS001A01T05.FP_PARAM.DampingTime" : Int AT %DB5045.DBW50, 500 ms
   "2915RS001A01T05.FP_PARAM.Force_Value" : Real AT %DB5045.DBD52, 500 ms
   "2915RS001A01T05.FP_PARAM.Scale_Min" : Real AT %DB5045.DBD56, 500 ms
   "2915RS001A01T05.FP_PARAM.Scale_Max" : Real AT %DB5045.DBD60, 500 ms
   "2915RS001A01T05.FP_PARAM.Gradient" : Real AT %DB5045.DBD64, 500 ms
   "2915RS001A01T05.FP_PARAM.Grad_Pos" : Real AT %DB5045.DBD68, 500 ms
   "2915RS001A01T05.FP_PARAM.Grad_Neg" : Real AT %DB5045.DBD72, 500 ms
   "2915RS001A01T05.FP_PARAM.Grad_X" : Real AT %DB5045.DBD76, 500 ms
   "2915RS001A01T05.FP_PARAM.Gradient_Time_Pre" : Int AT %DB5045.DBW80, 500 ms
   "2915RS001A01T05.FP_PARAM.Gradient_Time_ACC" : Int AT %DB5045.DBW82, 500 ms
   "2915RS001A01T05.FP_PARAM.Alarm_Hyst" : Real AT %DB5045.DBD84, 500 ms
   "2915RS001A01T05.FP_PARAM.AlarmLimit_H3" : Real AT %DB5045.DBD88, 500 ms
   "2915RS001A01T05.FP_PARAM.AlarmLimit_H2" : Real AT %DB5045.DBD92, 500 ms
   "2915RS001A01T05.FP_PARAM.AlarmLimit_H1" : Real AT %DB5045.DBD96, 500 ms
   "2915RS001A01T05.FP_PARAM.AlarmLimit_L1" : Real AT %DB5045.DBD100, 500 ms
   "2915RS001A01T05.FP_PARAM.AlarmLimit_L2" : Real AT %DB5045.DBD104, 500 ms
   "2915RS001A01T05.FP_PARAM.AlarmLimit_L3" : Real AT %DB5045.DBD108, 500 ms
   "2915RS001A01T05.FP_PARAM.AlarmDelay_H3_Pre" : Int AT %DB5045.DBW112, 500 ms
   "2915RS001A01T05.FP_PARAM.AlarmDelay_H3_Acc" : Int AT %DB5045.DBW114, 500 ms
   "2915RS001A01T05.FP_PARAM.AlarmDelay_H2_Pre" : Int AT %DB5045.DBW116, 500 ms
   "2915RS001A01T05.FP_PARAM.AlarmDelay_H2_Acc" : Int AT %DB5045.DBW118, 500 ms
   "2915RS001A01T05.FP_PARAM.AlarmDelay_H1_Pre" : Int AT %DB5045.DBW120, 500 ms
   "2915RS001A01T05.FP_PARAM.AlarmDelay_H1_Acc" : Int AT %DB5045.DBW122, 500 ms
   "2915RS001A01T05.FP_PARAM.AlarmDelay_L1_Pre" : Int AT %DB5045.DBW124, 500 ms
   "2915RS001A01T05.FP_PARAM.AlarmDelay_L1_Acc" : Int AT %DB5045.DBW126, 500 ms
   "2915RS001A01T05.FP_PARAM.AlarmDelay_L2_Pre" : Int AT %DB5045.DBW128, 500 ms
   "2915RS001A01T05.FP_PARAM.AlarmDelay_L2_Acc" : Int AT %DB5045.DBW130, 500 ms
   "2915RS001A01T05.FP_PARAM.AlarmDelay_L3_Pre" : Int AT %DB5045.DBW132, 500 ms
   "2915RS001A01T05.FP_PARAM.AlarmDelay_L3_Acc" : Int AT %DB5045.DBW134, 500 ms
   "2915RS001A01T05.FP_PARAM.OpenLoopDelay_Pre" : Int AT %DB5045.DBW136, 500 ms
   "2915RS001A01T05.FP_PARAM.OpenLoopDelay_Acc" : Int AT %DB5045.DBW138, 500 ms
   "2915RS001A01T05.FP_PARAM.OverRangeDelay_Pre" : Int AT %DB5045.DBW140, 500 ms
   "2915RS001A01T05.FP_PARAM.OverRangeDelay_Acc" : Int AT %DB5045.DBW142, 500 ms
   "2915RS001A01T05.FP_PARAM.AuxLimit_H2_Value" : Real AT %DB5045.DBD144, 500 ms
   "2915RS001A01T05.FP_PARAM.AuxLimit_H1_Value" : Real AT %DB5045.DBD148, 500 ms
   "2915RS001A01T05.FP_PARAM.AuxLimit_L2_Value" : Real AT %DB5045.DBD152, 500 ms
   "2915RS001A01T05.FP_PARAM.AuxLimit_L1_Value" : Real AT %DB5045.DBD156, 500 ms
   "2915RS001A01T05.Unit" : TextRef, internal   // Еденицы измерения При експорте из ECS через скрипт заполняется автоматически, если теги копируются в ручную то требуется задатать свойство Text
   "2915RS001A01T05.Decimals" : TextRef, internal   // Формат отображения При експорте из ECS через скрипт, заполняется автоматически. Если теги копируются в ручную то требуется задатать свойство Text s999999.9
   "2915RS001A01T05.FP_EN.Square" : Bool AT %DB5045.DBX46.0, 500 ms
   "2915RS001A01T05.FP_EN.SquareRoot" : Bool AT %DB5045.DBX46.1, 500 ms
   "2915RS001A01T05.FP_EN.ParentSupress" : Bool AT %DB5045.DBX46.2, 500 ms
   "2915RS001A01T05.FP_EN.ParentSupressUnit" : Bool AT %DB5045.DBX46.3, 500 ms
   "2915RS001A01T05.FP_EN.Force" : Bool AT %DB5045.DBX46.4, 500 ms
   "2915RS001A01T05.FP_EN.Damping" : Bool AT %DB5045.DBX46.5, 500 ms
   "2915RS001A01T05.FP_EN.Gradient_Pos" : Bool AT %DB5045.DBX46.6, 500 ms
   "2915RS001A01T05.FP_EN.Gradient_Neg" : Bool AT %DB5045.DBX46.7, 500 ms
   "2915RS001A01T05.FP_EN.Hysteresis" : Bool AT %DB5045.DBX47.0, 500 ms
   "2915RS001A01T05.FP_EN.Alarm_H3" : Bool AT %DB5045.DBX47.1, 500 ms
   "2915RS001A01T05.FP_EN.Alarm_H2" : Bool AT %DB5045.DBX47.2, 500 ms
   "2915RS001A01T05.FP_EN.Alarm_H1" : Bool AT %DB5045.DBX47.3, 500 ms
   "2915RS001A01T05.FP_EN.Alarm_L1" : Bool AT %DB5045.DBX47.4, 500 ms
   "2915RS001A01T05.FP_EN.Alarm_L2" : Bool AT %DB5045.DBX47.5, 500 ms
   "2915RS001A01T05.FP_EN.Alarm_L3" : Bool AT %DB5045.DBX47.6, 500 ms
   "2915RS001A01T05.FP_EN.AlarmDelay_H3" : Bool AT %DB5045.DBX47.7, 500 ms
   "2915RS001A01T05.FP_EN.AlarmDelay_H2" : Bool AT %DB5045.DBX48.0, 500 ms
   "2915RS001A01T05.FP_EN.AlarmDelay_H1" : Bool AT %DB5045.DBX48.1, 500 ms
   "2915RS001A01T05.FP_EN.AlarmDelay_L1" : Bool AT %DB5045.DBX48.2, 500 ms
   "2915RS001A01T05.FP_EN.AlarmDelay_L2" : Bool AT %DB5045.DBX48.3, 500 ms
   "2915RS001A01T05.FP_EN.AlarmDelay_L3" : Bool AT %DB5045.DBX48.4, 500 ms
   "2915RS001A01T05.FP_EN.ROC_Warn" : Bool AT %DB5045.DBX48.5, 500 ms
   "2915RS001A01T05.FP_EN.U_Range_Warn" : Bool AT %DB5045.DBX48.6, 500 ms
   "2915RS001A01T05.FP_EN.O_Range_Warn" : Bool AT %DB5045.DBX48.7, 500 ms
   "2915RS001A01T05.trend_tag_name" : TextRef, internal   // Еденицы измерения При експорте из ECS через скрипт - заполняется автоматически, если теги копируются в ручную то требуется задатать свойство Text - имя тега для тренда
   "2915RS001A01T05.DQ.AL_H3" : Bool AT %DB5045.DBX16.0, 500 ms
   "2915RS001A01T05.DQ.AL_H2" : Bool AT %DB5045.DBX16.1, 500 ms
   "2915RS001A01T05.DQ.AL_H1" : Bool AT %DB5045.DBX16.2, 500 ms
   "2915RS001A01T05.DQ.AL_L1" : Bool AT %DB5045.DBX16.3, 500 ms
   "2915RS001A01T05.DQ.AL_L2" : Bool AT %DB5045.DBX16.4, 500 ms
   "2915RS001A01T05.DQ.AL_L3" : Bool AT %DB5045.DBX16.5, 500 ms
   "2915RS001A01T05.DQ.SIG_OK" : Bool AT %DB5045.DBX16.6, 500 ms
   "2915RS001A01T05.DQ.LIM_H2" : Bool AT %DB5045.DBX16.7, 500 ms
   "2915RS001A01T05.DQ.LIM_H1" : Bool AT %DB5045.DBX17.0, 500 ms
   "2915RS001A01T05.DQ.LIM_L1" : Bool AT %DB5045.DBX17.1, 500 ms
   "2915RS001A01T05.DQ.LIM_L2" : Bool AT %DB5045.DBX17.2, 500 ms
   "2915RS001A01T05.DQ.GR_P" : Bool AT %DB5045.DBX17.3, 500 ms
   "2915RS001A01T05.DQ.GR_N" : Bool AT %DB5045.DBX17.4, 500 ms
   "2915RS001A01T05.I.IN" : Real AT %DB5045.DBD2, 500 ms
   "2915RS001A01T05.I.SIG_TYPE" : Int AT %DB5045.DBW0, 500 ms
   "2915RS001A01T05.I.FI_BUS" : Byte AT %DB5045.DBB6, 500 ms
   "2915RS001A01T05.DI.U_RANGE" : Bool AT %DB5045.DBX7.0, 500 ms
   "2915RS001A01T05.DI.O_RANGE" : Bool AT %DB5045.DBX7.1, 500 ms
   "2915RS001A01T05.DI.SIG_FAULT" : Bool AT %DB5045.DBX7.2, 500 ms
   "2915RS001A01T05.DI.EnConfig" : Bool AT %DB5045.DBX7.3, 500 ms
   "2915RS001A01T05.DI.AEN" : Bool AT %DB5045.DBX7.4, 500 ms
   "2915RS001A01T05.DI.AL_SUPR" : Bool AT %DB5045.DBX7.5, 500 ms
   "2915RS001A01T05.Q.PV_NORM" : Real AT %DB5045.DBD8, 500 ms
   "2915RS001A01T05.Q.PV_SCAL" : Real AT %DB5045.DBD12, 500 ms
   "2915RS001A01T05.ParentInfo" : TextRef, internal   // Имя родителя для попап окна, вкладка инфо. При експорте из ECS через скрипт заполняется автоматически, если теги копируются в ручную то требуется в ручную задатать свойство Start Value

HMI tags "2915RS001N01T01"
   "2915RS001N01T01.MSW" : 52809b66-421d-457f-8884-6f7a49d4e247 AT %DB5303.DBX18.0, 500 ms
   "2915RS001N01T01.DefaultText" : TextRef, internal   // Заголовок POPUP окна. При експорте из ECS через скрипт заполняется автоматически, если теги копируются в ручную то требуется в ручную задатать свойство Start Value
   "2915RS001N01T01.BlockInfo" : Array [0..2] of Int AT %DB5303.DBX38.0, 500 ms
   "2915RS001N01T01.StatusWork" : Int AT %DB5303.DBW242, 500 ms
   "2915RS001N01T01.FP_PARAM.DampingTime" : Int AT %DB5303.DBW50, 500 ms
   "2915RS001N01T01.FP_PARAM.Force_Value" : Real AT %DB5303.DBD52, 500 ms
   "2915RS001N01T01.FP_PARAM.Scale_Min" : Real AT %DB5303.DBD56, 500 ms
   "2915RS001N01T01.FP_PARAM.Scale_Max" : Real AT %DB5303.DBD60, 500 ms
   "2915RS001N01T01.FP_PARAM.Gradient" : Real AT %DB5303.DBD64, 500 ms
   "2915RS001N01T01.FP_PARAM.Grad_Pos" : Real AT %DB5303.DBD68, 500 ms
   "2915RS001N01T01.FP_PARAM.Grad_Neg" : Real AT %DB5303.DBD72, 500 ms
   "2915RS001N01T01.FP_PARAM.Grad_X" : Real AT %DB5303.DBD76, 500 ms
   "2915RS001N01T01.FP_PARAM.Gradient_Time_Pre" : Int AT %DB5303.DBW80, 500 ms
   "2915RS001N01T01.FP_PARAM.Gradient_Time_ACC" : Int AT %DB5303.DBW82, 500 ms
   "2915RS001N01T01.FP_PARAM.Alarm_Hyst" : Real AT %DB5303.DBD84, 500 ms
   "2915RS001N01T01.FP_PARAM.AlarmLimit_H3" : Real AT %DB5303.DBD88, 500 ms
   "2915RS001N01T01.FP_PARAM.AlarmLimit_H2" : Real AT %DB5303.DBD92, 500 ms
   "2915RS001N01T01.FP_PARAM.AlarmLimit_H1" : Real AT %DB5303.DBD96, 500 ms
   "2915RS001N01T01.FP_PARAM.AlarmLimit_L1" : Real AT %DB5303.DBD100, 500 ms
   "2915RS001N01T01.FP_PARAM.AlarmLimit_L2" : Real AT %DB5303.DBD104, 500 ms
   "2915RS001N01T01.FP_PARAM.AlarmLimit_L3" : Real AT %DB5303.DBD108, 500 ms
   "2915RS001N01T01.FP_PARAM.AlarmDelay_H3_Pre" : Int AT %DB5303.DBW112, 500 ms
   "2915RS001N01T01.FP_PARAM.AlarmDelay_H3_Acc" : Int AT %DB5303.DBW114, 500 ms
   "2915RS001N01T01.FP_PARAM.AlarmDelay_H2_Pre" : Int AT %DB5303.DBW116, 500 ms
   "2915RS001N01T01.FP_PARAM.AlarmDelay_H2_Acc" : Int AT %DB5303.DBW118, 500 ms
   "2915RS001N01T01.FP_PARAM.AlarmDelay_H1_Pre" : Int AT %DB5303.DBW120, 500 ms
   "2915RS001N01T01.FP_PARAM.AlarmDelay_H1_Acc" : Int AT %DB5303.DBW122, 500 ms
   "2915RS001N01T01.FP_PARAM.AlarmDelay_L1_Pre" : Int AT %DB5303.DBW124, 500 ms
   "2915RS001N01T01.FP_PARAM.AlarmDelay_L1_Acc" : Int AT %DB5303.DBW126, 500 ms
   "2915RS001N01T01.FP_PARAM.AlarmDelay_L2_Pre" : Int AT %DB5303.DBW128, 500 ms
   "2915RS001N01T01.FP_PARAM.AlarmDelay_L2_Acc" : Int AT %DB5303.DBW130, 500 ms
   "2915RS001N01T01.FP_PARAM.AlarmDelay_L3_Pre" : Int AT %DB5303.DBW132, 500 ms
   "2915RS001N01T01.FP_PARAM.AlarmDelay_L3_Acc" : Int AT %DB5303.DBW134, 500 ms
   "2915RS001N01T01.FP_PARAM.OpenLoopDelay_Pre" : Int AT %DB5303.DBW136, 500 ms
   "2915RS001N01T01.FP_PARAM.OpenLoopDelay_Acc" : Int AT %DB5303.DBW138, 500 ms
   "2915RS001N01T01.FP_PARAM.OverRangeDelay_Pre" : Int AT %DB5303.DBW140, 500 ms
   "2915RS001N01T01.FP_PARAM.OverRangeDelay_Acc" : Int AT %DB5303.DBW142, 500 ms
   "2915RS001N01T01.FP_PARAM.AuxLimit_H2_Value" : Real AT %DB5303.DBD144, 500 ms
   "2915RS001N01T01.FP_PARAM.AuxLimit_H1_Value" : Real AT %DB5303.DBD148, 500 ms
   "2915RS001N01T01.FP_PARAM.AuxLimit_L2_Value" : Real AT %DB5303.DBD152, 500 ms
   "2915RS001N01T01.FP_PARAM.AuxLimit_L1_Value" : Real AT %DB5303.DBD156, 500 ms
   "2915RS001N01T01.Unit" : TextRef, internal   // Еденицы измерения При експорте из ECS через скрипт заполняется автоматически, если теги копируются в ручную то требуется задатать свойство Text
   "2915RS001N01T01.Decimals" : TextRef, internal   // Формат отображения При експорте из ECS через скрипт, заполняется автоматически. Если теги копируются в ручную то требуется задатать свойство Text s999999.9
   "2915RS001N01T01.FP_EN.Square" : Bool AT %DB5303.DBX46.0, 500 ms
   "2915RS001N01T01.FP_EN.SquareRoot" : Bool AT %DB5303.DBX46.1, 500 ms
   "2915RS001N01T01.FP_EN.ParentSupress" : Bool AT %DB5303.DBX46.2, 500 ms
   "2915RS001N01T01.FP_EN.ParentSupressUnit" : Bool AT %DB5303.DBX46.3, 500 ms
   "2915RS001N01T01.FP_EN.Force" : Bool AT %DB5303.DBX46.4, 500 ms
   "2915RS001N01T01.FP_EN.Damping" : Bool AT %DB5303.DBX46.5, 500 ms
   "2915RS001N01T01.FP_EN.Gradient_Pos" : Bool AT %DB5303.DBX46.6, 500 ms
   "2915RS001N01T01.FP_EN.Gradient_Neg" : Bool AT %DB5303.DBX46.7, 500 ms
   "2915RS001N01T01.FP_EN.Hysteresis" : Bool AT %DB5303.DBX47.0, 500 ms
   "2915RS001N01T01.FP_EN.Alarm_H3" : Bool AT %DB5303.DBX47.1, 500 ms
   "2915RS001N01T01.FP_EN.Alarm_H2" : Bool AT %DB5303.DBX47.2, 500 ms
   "2915RS001N01T01.FP_EN.Alarm_H1" : Bool AT %DB5303.DBX47.3, 500 ms
   "2915RS001N01T01.FP_EN.Alarm_L1" : Bool AT %DB5303.DBX47.4, 500 ms
   "2915RS001N01T01.FP_EN.Alarm_L2" : Bool AT %DB5303.DBX47.5, 500 ms
   "2915RS001N01T01.FP_EN.Alarm_L3" : Bool AT %DB5303.DBX47.6, 500 ms
   "2915RS001N01T01.FP_EN.AlarmDelay_H3" : Bool AT %DB5303.DBX47.7, 500 ms
   "2915RS001N01T01.FP_EN.AlarmDelay_H2" : Bool AT %DB5303.DBX48.0, 500 ms
   "2915RS001N01T01.FP_EN.AlarmDelay_H1" : Bool AT %DB5303.DBX48.1, 500 ms
   "2915RS001N01T01.FP_EN.AlarmDelay_L1" : Bool AT %DB5303.DBX48.2, 500 ms
   "2915RS001N01T01.FP_EN.AlarmDelay_L2" : Bool AT %DB5303.DBX48.3, 500 ms
   "2915RS001N01T01.FP_EN.AlarmDelay_L3" : Bool AT %DB5303.DBX48.4, 500 ms
   "2915RS001N01T01.FP_EN.ROC_Warn" : Bool AT %DB5303.DBX48.5, 500 ms
   "2915RS001N01T01.FP_EN.U_Range_Warn" : Bool AT %DB5303.DBX48.6, 500 ms
   "2915RS001N01T01.FP_EN.O_Range_Warn" : Bool AT %DB5303.DBX48.7, 500 ms
   "2915RS001N01T01.trend_tag_name" : TextRef, internal   // Еденицы измерения При експорте из ECS через скрипт - заполняется автоматически, если теги копируются в ручную то требуется задатать свойство Text - имя тега для тренда
   "2915RS001N01T01.DQ.AL_H3" : Bool AT %DB5303.DBX16.0, 500 ms
   "2915RS001N01T01.DQ.AL_H2" : Bool AT %DB5303.DBX16.1, 500 ms
   "2915RS001N01T01.DQ.AL_H1" : Bool AT %DB5303.DBX16.2, 500 ms
   "2915RS001N01T01.DQ.AL_L1" : Bool AT %DB5303.DBX16.3, 500 ms
   "2915RS001N01T01.DQ.AL_L2" : Bool AT %DB5303.DBX16.4, 500 ms
   "2915RS001N01T01.DQ.AL_L3" : Bool AT %DB5303.DBX16.5, 500 ms
   "2915RS001N01T01.DQ.SIG_OK" : Bool AT %DB5303.DBX16.6, 500 ms
   "2915RS001N01T01.DQ.LIM_H2" : Bool AT %DB5303.DBX16.7, 500 ms
   "2915RS001N01T01.DQ.LIM_H1" : Bool AT %DB5303.DBX17.0, 500 ms
   "2915RS001N01T01.DQ.LIM_L1" : Bool AT %DB5303.DBX17.1, 500 ms
   "2915RS001N01T01.DQ.LIM_L2" : Bool AT %DB5303.DBX17.2, 500 ms
   "2915RS001N01T01.DQ.GR_P" : Bool AT %DB5303.DBX17.3, 500 ms
   "2915RS001N01T01.DQ.GR_N" : Bool AT %DB5303.DBX17.4, 500 ms
   "2915RS001N01T01.I.IN" : Real AT %DB5303.DBD2, 500 ms
   "2915RS001N01T01.I.SIG_TYPE" : Int AT %DB5303.DBW0, 500 ms
   "2915RS001N01T01.I.FI_BUS" : Byte AT %DB5303.DBB6, 500 ms
   "2915RS001N01T01.DI.U_RANGE" : Bool AT %DB5303.DBX7.0, 500 ms
   "2915RS001N01T01.DI.O_RANGE" : Bool AT %DB5303.DBX7.1, 500 ms
   "2915RS001N01T01.DI.SIG_FAULT" : Bool AT %DB5303.DBX7.2, 500 ms
   "2915RS001N01T01.DI.EnConfig" : Bool AT %DB5303.DBX7.3, 500 ms
   "2915RS001N01T01.DI.AEN" : Bool AT %DB5303.DBX7.4, 500 ms
   "2915RS001N01T01.DI.AL_SUPR" : Bool AT %DB5303.DBX7.5, 500 ms
   "2915RS001N01T01.Q.PV_NORM" : Real AT %DB5303.DBD8, 500 ms
   "2915RS001N01T01.Q.PV_SCAL" : Real AT %DB5303.DBD12, 500 ms
   "2915RS001N01T01.ParentInfo" : TextRef, internal   // Имя родителя для попап окна, вкладка инфо. При експорте из ECS через скрипт заполняется автоматически, если теги копируются в ручную то требуется в ручную задатать свойство Start Value

HMI tags "2920RS001A01A01"
   "2920RS001A01A01.MSW" : 52809b66-421d-457f-8884-6f7a49d4e247 AT %DB5046.DBX18.0, 500 ms
   "2920RS001A01A01.DefaultText" : TextRef, internal   // Заголовок POPUP окна. При експорте из ECS через скрипт заполняется автоматически, если теги копируются в ручную то требуется в ручную задатать свойство Start Value
   "2920RS001A01A01.BlockInfo" : Array [0..2] of Int AT %DB5046.DBX38.0, 500 ms
   "2920RS001A01A01.StatusWork" : Int AT %DB5046.DBW242, 500 ms
   "2920RS001A01A01.FP_PARAM.DampingTime" : Int AT %DB5046.DBW50, 500 ms
   "2920RS001A01A01.FP_PARAM.Force_Value" : Real AT %DB5046.DBD52, 500 ms
   "2920RS001A01A01.FP_PARAM.Scale_Min" : Real AT %DB5046.DBD56, 500 ms
   "2920RS001A01A01.FP_PARAM.Scale_Max" : Real AT %DB5046.DBD60, 500 ms
   "2920RS001A01A01.FP_PARAM.Gradient" : Real AT %DB5046.DBD64, 500 ms
   "2920RS001A01A01.FP_PARAM.Grad_Pos" : Real AT %DB5046.DBD68, 500 ms
   "2920RS001A01A01.FP_PARAM.Grad_Neg" : Real AT %DB5046.DBD72, 500 ms
   "2920RS001A01A01.FP_PARAM.Grad_X" : Real AT %DB5046.DBD76, 500 ms
   "2920RS001A01A01.FP_PARAM.Gradient_Time_Pre" : Int AT %DB5046.DBW80, 500 ms
   "2920RS001A01A01.FP_PARAM.Gradient_Time_ACC" : Int AT %DB5046.DBW82, 500 ms
   "2920RS001A01A01.FP_PARAM.Alarm_Hyst" : Real AT %DB5046.DBD84, 500 ms
   "2920RS001A01A01.FP_PARAM.AlarmLimit_H3" : Real AT %DB5046.DBD88, 500 ms
   "2920RS001A01A01.FP_PARAM.AlarmLimit_H2" : Real AT %DB5046.DBD92, 500 ms
   "2920RS001A01A01.FP_PARAM.AlarmLimit_H1" : Real AT %DB5046.DBD96, 500 ms
   "2920RS001A01A01.FP_PARAM.AlarmLimit_L1" : Real AT %DB5046.DBD100, 500 ms
   "2920RS001A01A01.FP_PARAM.AlarmLimit_L2" : Real AT %DB5046.DBD104, 500 ms
   "2920RS001A01A01.FP_PARAM.AlarmLimit_L3" : Real AT %DB5046.DBD108, 500 ms
   "2920RS001A01A01.FP_PARAM.AlarmDelay_H3_Pre" : Int AT %DB5046.DBW112, 500 ms
   "2920RS001A01A01.FP_PARAM.AlarmDelay_H3_Acc" : Int AT %DB5046.DBW114, 500 ms
   "2920RS001A01A01.FP_PARAM.AlarmDelay_H2_Pre" : Int AT %DB5046.DBW116, 500 ms
   "2920RS001A01A01.FP_PARAM.AlarmDelay_H2_Acc" : Int AT %DB5046.DBW118, 500 ms
   "2920RS001A01A01.FP_PARAM.AlarmDelay_H1_Pre" : Int AT %DB5046.DBW120, 500 ms
   "2920RS001A01A01.FP_PARAM.AlarmDelay_H1_Acc" : Int AT %DB5046.DBW122, 500 ms
   "2920RS001A01A01.FP_PARAM.AlarmDelay_L1_Pre" : Int AT %DB5046.DBW124, 500 ms
   "2920RS001A01A01.FP_PARAM.AlarmDelay_L1_Acc" : Int AT %DB5046.DBW126, 500 ms
   "2920RS001A01A01.FP_PARAM.AlarmDelay_L2_Pre" : Int AT %DB5046.DBW128, 500 ms
   "2920RS001A01A01.FP_PARAM.AlarmDelay_L2_Acc" : Int AT %DB5046.DBW130, 500 ms
   "2920RS001A01A01.FP_PARAM.AlarmDelay_L3_Pre" : Int AT %DB5046.DBW132, 500 ms
   "2920RS001A01A01.FP_PARAM.AlarmDelay_L3_Acc" : Int AT %DB5046.DBW134, 500 ms
   "2920RS001A01A01.FP_PARAM.OpenLoopDelay_Pre" : Int AT %DB5046.DBW136, 500 ms
   "2920RS001A01A01.FP_PARAM.OpenLoopDelay_Acc" : Int AT %DB5046.DBW138, 500 ms
   "2920RS001A01A01.FP_PARAM.OverRangeDelay_Pre" : Int AT %DB5046.DBW140, 500 ms
   "2920RS001A01A01.FP_PARAM.OverRangeDelay_Acc" : Int AT %DB5046.DBW142, 500 ms
   "2920RS001A01A01.FP_PARAM.AuxLimit_H2_Value" : Real AT %DB5046.DBD144, 500 ms
   "2920RS001A01A01.FP_PARAM.AuxLimit_H1_Value" : Real AT %DB5046.DBD148, 500 ms
   "2920RS001A01A01.FP_PARAM.AuxLimit_L2_Value" : Real AT %DB5046.DBD152, 500 ms
   "2920RS001A01A01.FP_PARAM.AuxLimit_L1_Value" : Real AT %DB5046.DBD156, 500 ms
   "2920RS001A01A01.Unit" : TextRef, internal   // Еденицы измерения При експорте из ECS через скрипт заполняется автоматически, если теги копируются в ручную то требуется задатать свойство Text
   "2920RS001A01A01.Decimals" : TextRef, internal   // Формат отображения При експорте из ECS через скрипт, заполняется автоматически. Если теги копируются в ручную то требуется задатать свойство Text s999999.9
   "2920RS001A01A01.FP_EN.Square" : Bool AT %DB5046.DBX46.0, 500 ms
   "2920RS001A01A01.FP_EN.SquareRoot" : Bool AT %DB5046.DBX46.1, 500 ms
   "2920RS001A01A01.FP_EN.ParentSupress" : Bool AT %DB5046.DBX46.2, 500 ms
   "2920RS001A01A01.FP_EN.ParentSupressUnit" : Bool AT %DB5046.DBX46.3, 500 ms
   "2920RS001A01A01.FP_EN.Force" : Bool AT %DB5046.DBX46.4, 500 ms
   "2920RS001A01A01.FP_EN.Damping" : Bool AT %DB5046.DBX46.5, 500 ms
   "2920RS001A01A01.FP_EN.Gradient_Pos" : Bool AT %DB5046.DBX46.6, 500 ms
   "2920RS001A01A01.FP_EN.Gradient_Neg" : Bool AT %DB5046.DBX46.7, 500 ms
   "2920RS001A01A01.FP_EN.Hysteresis" : Bool AT %DB5046.DBX47.0, 500 ms
   "2920RS001A01A01.FP_EN.Alarm_H3" : Bool AT %DB5046.DBX47.1, 500 ms
   "2920RS001A01A01.FP_EN.Alarm_H2" : Bool AT %DB5046.DBX47.2, 500 ms
   "2920RS001A01A01.FP_EN.Alarm_H1" : Bool AT %DB5046.DBX47.3, 500 ms
   "2920RS001A01A01.FP_EN.Alarm_L1" : Bool AT %DB5046.DBX47.4, 500 ms
   "2920RS001A01A01.FP_EN.Alarm_L2" : Bool AT %DB5046.DBX47.5, 500 ms
   "2920RS001A01A01.FP_EN.Alarm_L3" : Bool AT %DB5046.DBX47.6, 500 ms
   "2920RS001A01A01.FP_EN.AlarmDelay_H3" : Bool AT %DB5046.DBX47.7, 500 ms
   "2920RS001A01A01.FP_EN.AlarmDelay_H2" : Bool AT %DB5046.DBX48.0, 500 ms
   "2920RS001A01A01.FP_EN.AlarmDelay_H1" : Bool AT %DB5046.DBX48.1, 500 ms
   "2920RS001A01A01.FP_EN.AlarmDelay_L1" : Bool AT %DB5046.DBX48.2, 500 ms
   "2920RS001A01A01.FP_EN.AlarmDelay_L2" : Bool AT %DB5046.DBX48.3, 500 ms
   "2920RS001A01A01.FP_EN.AlarmDelay_L3" : Bool AT %DB5046.DBX48.4, 500 ms
   "2920RS001A01A01.FP_EN.ROC_Warn" : Bool AT %DB5046.DBX48.5, 500 ms
   "2920RS001A01A01.FP_EN.U_Range_Warn" : Bool AT %DB5046.DBX48.6, 500 ms
   "2920RS001A01A01.FP_EN.O_Range_Warn" : Bool AT %DB5046.DBX48.7, 500 ms
   "2920RS001A01A01.trend_tag_name" : TextRef, internal   // Еденицы измерения При експорте из ECS через скрипт - заполняется автоматически, если теги копируются в ручную то требуется задатать свойство Text - имя тега для тренда
   "2920RS001A01A01.DQ.AL_H3" : Bool AT %DB5046.DBX16.0, 500 ms
   "2920RS001A01A01.DQ.AL_H2" : Bool AT %DB5046.DBX16.1, 500 ms
   "2920RS001A01A01.DQ.AL_H1" : Bool AT %DB5046.DBX16.2, 500 ms
   "2920RS001A01A01.DQ.AL_L1" : Bool AT %DB5046.DBX16.3, 500 ms
   "2920RS001A01A01.DQ.AL_L2" : Bool AT %DB5046.DBX16.4, 500 ms
   "2920RS001A01A01.DQ.AL_L3" : Bool AT %DB5046.DBX16.5, 500 ms
   "2920RS001A01A01.DQ.SIG_OK" : Bool AT %DB5046.DBX16.6, 500 ms
   "2920RS001A01A01.DQ.LIM_H2" : Bool AT %DB5046.DBX16.7, 500 ms
   "2920RS001A01A01.DQ.LIM_H1" : Bool AT %DB5046.DBX17.0, 500 ms
   "2920RS001A01A01.DQ.LIM_L1" : Bool AT %DB5046.DBX17.1, 500 ms
   "2920RS001A01A01.DQ.LIM_L2" : Bool AT %DB5046.DBX17.2, 500 ms
   "2920RS001A01A01.DQ.GR_P" : Bool AT %DB5046.DBX17.3, 500 ms
   "2920RS001A01A01.DQ.GR_N" : Bool AT %DB5046.DBX17.4, 500 ms
   "2920RS001A01A01.I.IN" : Real AT %DB5046.DBD2, 500 ms
   "2920RS001A01A01.I.SIG_TYPE" : Int AT %DB5046.DBW0, 500 ms
   "2920RS001A01A01.I.FI_BUS" : Byte AT %DB5046.DBB6, 500 ms
   "2920RS001A01A01.DI.U_RANGE" : Bool AT %DB5046.DBX7.0, 500 ms
   "2920RS001A01A01.DI.O_RANGE" : Bool AT %DB5046.DBX7.1, 500 ms
   "2920RS001A01A01.DI.SIG_FAULT" : Bool AT %DB5046.DBX7.2, 500 ms
   "2920RS001A01A01.DI.EnConfig" : Bool AT %DB5046.DBX7.3, 500 ms
   "2920RS001A01A01.DI.AEN" : Bool AT %DB5046.DBX7.4, 500 ms
   "2920RS001A01A01.DI.AL_SUPR" : Bool AT %DB5046.DBX7.5, 500 ms
   "2920RS001A01A01.Q.PV_NORM" : Real AT %DB5046.DBD8, 500 ms
   "2920RS001A01A01.Q.PV_SCAL" : Real AT %DB5046.DBD12, 500 ms
   "2920RS001A01A01.ParentInfo" : TextRef, internal   // Имя родителя для попап окна, вкладка инфо. При експорте из ECS через скрипт заполняется автоматически, если теги копируются в ручную то требуется в ручную задатать свойство Start Value

HMI tags "2920RS001A01A02"
   "2920RS001A01A02.MSW" : 52809b66-421d-457f-8884-6f7a49d4e247 AT %DB5047.DBX18.0, 500 ms
   "2920RS001A01A02.DefaultText" : TextRef, internal   // Заголовок POPUP окна. При експорте из ECS через скрипт заполняется автоматически, если теги копируются в ручную то требуется в ручную задатать свойство Start Value
   "2920RS001A01A02.BlockInfo" : Array [0..2] of Int AT %DB5047.DBX38.0, 500 ms
   "2920RS001A01A02.StatusWork" : Int AT %DB5047.DBW242, 500 ms
   "2920RS001A01A02.FP_PARAM.DampingTime" : Int AT %DB5047.DBW50, 500 ms
   "2920RS001A01A02.FP_PARAM.Force_Value" : Real AT %DB5047.DBD52, 500 ms
   "2920RS001A01A02.FP_PARAM.Scale_Min" : Real AT %DB5047.DBD56, 500 ms
   "2920RS001A01A02.FP_PARAM.Scale_Max" : Real AT %DB5047.DBD60, 500 ms
   "2920RS001A01A02.FP_PARAM.Gradient" : Real AT %DB5047.DBD64, 500 ms
   "2920RS001A01A02.FP_PARAM.Grad_Pos" : Real AT %DB5047.DBD68, 500 ms
   "2920RS001A01A02.FP_PARAM.Grad_Neg" : Real AT %DB5047.DBD72, 500 ms
   "2920RS001A01A02.FP_PARAM.Grad_X" : Real AT %DB5047.DBD76, 500 ms
   "2920RS001A01A02.FP_PARAM.Gradient_Time_Pre" : Int AT %DB5047.DBW80, 500 ms
   "2920RS001A01A02.FP_PARAM.Gradient_Time_ACC" : Int AT %DB5047.DBW82, 500 ms
   "2920RS001A01A02.FP_PARAM.Alarm_Hyst" : Real AT %DB5047.DBD84, 500 ms
   "2920RS001A01A02.FP_PARAM.AlarmLimit_H3" : Real AT %DB5047.DBD88, 500 ms
   "2920RS001A01A02.FP_PARAM.AlarmLimit_H2" : Real AT %DB5047.DBD92, 500 ms
   "2920RS001A01A02.FP_PARAM.AlarmLimit_H1" : Real AT %DB5047.DBD96, 500 ms
   "2920RS001A01A02.FP_PARAM.AlarmLimit_L1" : Real AT %DB5047.DBD100, 500 ms
   "2920RS001A01A02.FP_PARAM.AlarmLimit_L2" : Real AT %DB5047.DBD104, 500 ms
   "2920RS001A01A02.FP_PARAM.AlarmLimit_L3" : Real AT %DB5047.DBD108, 500 ms
   "2920RS001A01A02.FP_PARAM.AlarmDelay_H3_Pre" : Int AT %DB5047.DBW112, 500 ms
   "2920RS001A01A02.FP_PARAM.AlarmDelay_H3_Acc" : Int AT %DB5047.DBW114, 500 ms
   "2920RS001A01A02.FP_PARAM.AlarmDelay_H2_Pre" : Int AT %DB5047.DBW116, 500 ms
   "2920RS001A01A02.FP_PARAM.AlarmDelay_H2_Acc" : Int AT %DB5047.DBW118, 500 ms
   "2920RS001A01A02.FP_PARAM.AlarmDelay_H1_Pre" : Int AT %DB5047.DBW120, 500 ms
   "2920RS001A01A02.FP_PARAM.AlarmDelay_H1_Acc" : Int AT %DB5047.DBW122, 500 ms
   "2920RS001A01A02.FP_PARAM.AlarmDelay_L1_Pre" : Int AT %DB5047.DBW124, 500 ms
   "2920RS001A01A02.FP_PARAM.AlarmDelay_L1_Acc" : Int AT %DB5047.DBW126, 500 ms
   "2920RS001A01A02.FP_PARAM.AlarmDelay_L2_Pre" : Int AT %DB5047.DBW128, 500 ms
   "2920RS001A01A02.FP_PARAM.AlarmDelay_L2_Acc" : Int AT %DB5047.DBW130, 500 ms
   "2920RS001A01A02.FP_PARAM.AlarmDelay_L3_Pre" : Int AT %DB5047.DBW132, 500 ms
   "2920RS001A01A02.FP_PARAM.AlarmDelay_L3_Acc" : Int AT %DB5047.DBW134, 500 ms
   "2920RS001A01A02.FP_PARAM.OpenLoopDelay_Pre" : Int AT %DB5047.DBW136, 500 ms
   "2920RS001A01A02.FP_PARAM.OpenLoopDelay_Acc" : Int AT %DB5047.DBW138, 500 ms
   "2920RS001A01A02.FP_PARAM.OverRangeDelay_Pre" : Int AT %DB5047.DBW140, 500 ms
   "2920RS001A01A02.FP_PARAM.OverRangeDelay_Acc" : Int AT %DB5047.DBW142, 500 ms
   "2920RS001A01A02.FP_PARAM.AuxLimit_H2_Value" : Real AT %DB5047.DBD144, 500 ms
   "2920RS001A01A02.FP_PARAM.AuxLimit_H1_Value" : Real AT %DB5047.DBD148, 500 ms
   "2920RS001A01A02.FP_PARAM.AuxLimit_L2_Value" : Real AT %DB5047.DBD152, 500 ms
   "2920RS001A01A02.FP_PARAM.AuxLimit_L1_Value" : Real AT %DB5047.DBD156, 500 ms
   "2920RS001A01A02.Unit" : TextRef, internal   // Еденицы измерения При експорте из ECS через скрипт заполняется автоматически, если теги копируются в ручную то требуется задатать свойство Text
   "2920RS001A01A02.Decimals" : TextRef, internal   // Формат отображения При експорте из ECS через скрипт, заполняется автоматически. Если теги копируются в ручную то требуется задатать свойство Text s999999.9
   "2920RS001A01A02.FP_EN.Square" : Bool AT %DB5047.DBX46.0, 500 ms
   "2920RS001A01A02.FP_EN.SquareRoot" : Bool AT %DB5047.DBX46.1, 500 ms
   "2920RS001A01A02.FP_EN.ParentSupress" : Bool AT %DB5047.DBX46.2, 500 ms
   "2920RS001A01A02.FP_EN.ParentSupressUnit" : Bool AT %DB5047.DBX46.3, 500 ms
   "2920RS001A01A02.FP_EN.Force" : Bool AT %DB5047.DBX46.4, 500 ms
   "2920RS001A01A02.FP_EN.Damping" : Bool AT %DB5047.DBX46.5, 500 ms
   "2920RS001A01A02.FP_EN.Gradient_Pos" : Bool AT %DB5047.DBX46.6, 500 ms
   "2920RS001A01A02.FP_EN.Gradient_Neg" : Bool AT %DB5047.DBX46.7, 500 ms
   "2920RS001A01A02.FP_EN.Hysteresis" : Bool AT %DB5047.DBX47.0, 500 ms
   "2920RS001A01A02.FP_EN.Alarm_H3" : Bool AT %DB5047.DBX47.1, 500 ms
   "2920RS001A01A02.FP_EN.Alarm_H2" : Bool AT %DB5047.DBX47.2, 500 ms
   "2920RS001A01A02.FP_EN.Alarm_H1" : Bool AT %DB5047.DBX47.3, 500 ms
   "2920RS001A01A02.FP_EN.Alarm_L1" : Bool AT %DB5047.DBX47.4, 500 ms
   "2920RS001A01A02.FP_EN.Alarm_L2" : Bool AT %DB5047.DBX47.5, 500 ms
   "2920RS001A01A02.FP_EN.Alarm_L3" : Bool AT %DB5047.DBX47.6, 500 ms
   "2920RS001A01A02.FP_EN.AlarmDelay_H3" : Bool AT %DB5047.DBX47.7, 500 ms
   "2920RS001A01A02.FP_EN.AlarmDelay_H2" : Bool AT %DB5047.DBX48.0, 500 ms
   "2920RS001A01A02.FP_EN.AlarmDelay_H1" : Bool AT %DB5047.DBX48.1, 500 ms
   "2920RS001A01A02.FP_EN.AlarmDelay_L1" : Bool AT %DB5047.DBX48.2, 500 ms
   "2920RS001A01A02.FP_EN.AlarmDelay_L2" : Bool AT %DB5047.DBX48.3, 500 ms
   "2920RS001A01A02.FP_EN.AlarmDelay_L3" : Bool AT %DB5047.DBX48.4, 500 ms
   "2920RS001A01A02.FP_EN.ROC_Warn" : Bool AT %DB5047.DBX48.5, 500 ms
   "2920RS001A01A02.FP_EN.U_Range_Warn" : Bool AT %DB5047.DBX48.6, 500 ms
   "2920RS001A01A02.FP_EN.O_Range_Warn" : Bool AT %DB5047.DBX48.7, 500 ms
   "2920RS001A01A02.trend_tag_name" : TextRef, internal   // Еденицы измерения При експорте из ECS через скрипт - заполняется автоматически, если теги копируются в ручную то требуется задатать свойство Text - имя тега для тренда
   "2920RS001A01A02.DQ.AL_H3" : Bool AT %DB5047.DBX16.0, 500 ms
   "2920RS001A01A02.DQ.AL_H2" : Bool AT %DB5047.DBX16.1, 500 ms
   "2920RS001A01A02.DQ.AL_H1" : Bool AT %DB5047.DBX16.2, 500 ms
   "2920RS001A01A02.DQ.AL_L1" : Bool AT %DB5047.DBX16.3, 500 ms
   "2920RS001A01A02.DQ.AL_L2" : Bool AT %DB5047.DBX16.4, 500 ms
   "2920RS001A01A02.DQ.AL_L3" : Bool AT %DB5047.DBX16.5, 500 ms
   "2920RS001A01A02.DQ.SIG_OK" : Bool AT %DB5047.DBX16.6, 500 ms
   "2920RS001A01A02.DQ.LIM_H2" : Bool AT %DB5047.DBX16.7, 500 ms
   "2920RS001A01A02.DQ.LIM_H1" : Bool AT %DB5047.DBX17.0, 500 ms
   "2920RS001A01A02.DQ.LIM_L1" : Bool AT %DB5047.DBX17.1, 500 ms
   "2920RS001A01A02.DQ.LIM_L2" : Bool AT %DB5047.DBX17.2, 500 ms
   "2920RS001A01A02.DQ.GR_P" : Bool AT %DB5047.DBX17.3, 500 ms
   "2920RS001A01A02.DQ.GR_N" : Bool AT %DB5047.DBX17.4, 500 ms
   "2920RS001A01A02.I.IN" : Real AT %DB5047.DBD2, 500 ms
   "2920RS001A01A02.I.SIG_TYPE" : Int AT %DB5047.DBW0, 500 ms
   "2920RS001A01A02.I.FI_BUS" : Byte AT %DB5047.DBB6, 500 ms
   "2920RS001A01A02.DI.U_RANGE" : Bool AT %DB5047.DBX7.0, 500 ms
   "2920RS001A01A02.DI.O_RANGE" : Bool AT %DB5047.DBX7.1, 500 ms
   "2920RS001A01A02.DI.SIG_FAULT" : Bool AT %DB5047.DBX7.2, 500 ms
   "2920RS001A01A02.DI.EnConfig" : Bool AT %DB5047.DBX7.3, 500 ms
   "2920RS001A01A02.DI.AEN" : Bool AT %DB5047.DBX7.4, 500 ms
   "2920RS001A01A02.DI.AL_SUPR" : Bool AT %DB5047.DBX7.5, 500 ms
   "2920RS001A01A02.Q.PV_NORM" : Real AT %DB5047.DBD8, 500 ms
   "2920RS001A01A02.Q.PV_SCAL" : Real AT %DB5047.DBD12, 500 ms
   "2920RS001A01A02.ParentInfo" : TextRef, internal   // Имя родителя для попап окна, вкладка инфо. При експорте из ECS через скрипт заполняется автоматически, если теги копируются в ручную то требуется в ручную задатать свойство Start Value

HMI tags "2920RS001A01F01"
   "2920RS001A01F01.MSW" : 52809b66-421d-457f-8884-6f7a49d4e247 AT %DB5048.DBX18.0, 500 ms
   "2920RS001A01F01.DefaultText" : TextRef, internal   // Заголовок POPUP окна. При експорте из ECS через скрипт заполняется автоматически, если теги копируются в ручную то требуется в ручную задатать свойство Start Value
   "2920RS001A01F01.BlockInfo" : Array [0..2] of Int AT %DB5048.DBX38.0, 500 ms
   "2920RS001A01F01.StatusWork" : Int AT %DB5048.DBW242, 500 ms
   "2920RS001A01F01.FP_PARAM.DampingTime" : Int AT %DB5048.DBW50, 500 ms
   "2920RS001A01F01.FP_PARAM.Force_Value" : Real AT %DB5048.DBD52, 500 ms
   "2920RS001A01F01.FP_PARAM.Scale_Min" : Real AT %DB5048.DBD56, 500 ms
   "2920RS001A01F01.FP_PARAM.Scale_Max" : Real AT %DB5048.DBD60, 500 ms
   "2920RS001A01F01.FP_PARAM.Gradient" : Real AT %DB5048.DBD64, 500 ms
   "2920RS001A01F01.FP_PARAM.Grad_Pos" : Real AT %DB5048.DBD68, 500 ms
   "2920RS001A01F01.FP_PARAM.Grad_Neg" : Real AT %DB5048.DBD72, 500 ms
   "2920RS001A01F01.FP_PARAM.Grad_X" : Real AT %DB5048.DBD76, 500 ms
   "2920RS001A01F01.FP_PARAM.Gradient_Time_Pre" : Int AT %DB5048.DBW80, 500 ms
   "2920RS001A01F01.FP_PARAM.Gradient_Time_ACC" : Int AT %DB5048.DBW82, 500 ms
   "2920RS001A01F01.FP_PARAM.Alarm_Hyst" : Real AT %DB5048.DBD84, 500 ms
   "2920RS001A01F01.FP_PARAM.AlarmLimit_H3" : Real AT %DB5048.DBD88, 500 ms
   "2920RS001A01F01.FP_PARAM.AlarmLimit_H2" : Real AT %DB5048.DBD92, 500 ms
   "2920RS001A01F01.FP_PARAM.AlarmLimit_H1" : Real AT %DB5048.DBD96, 500 ms
   "2920RS001A01F01.FP_PARAM.AlarmLimit_L1" : Real AT %DB5048.DBD100, 500 ms
   "2920RS001A01F01.FP_PARAM.AlarmLimit_L2" : Real AT %DB5048.DBD104, 500 ms
   "2920RS001A01F01.FP_PARAM.AlarmLimit_L3" : Real AT %DB5048.DBD108, 500 ms
   "2920RS001A01F01.FP_PARAM.AlarmDelay_H3_Pre" : Int AT %DB5048.DBW112, 500 ms
   "2920RS001A01F01.FP_PARAM.AlarmDelay_H3_Acc" : Int AT %DB5048.DBW114, 500 ms
   "2920RS001A01F01.FP_PARAM.AlarmDelay_H2_Pre" : Int AT %DB5048.DBW116, 500 ms
   "2920RS001A01F01.FP_PARAM.AlarmDelay_H2_Acc" : Int AT %DB5048.DBW118, 500 ms
   "2920RS001A01F01.FP_PARAM.AlarmDelay_H1_Pre" : Int AT %DB5048.DBW120, 500 ms
   "2920RS001A01F01.FP_PARAM.AlarmDelay_H1_Acc" : Int AT %DB5048.DBW122, 500 ms
   "2920RS001A01F01.FP_PARAM.AlarmDelay_L1_Pre" : Int AT %DB5048.DBW124, 500 ms
   "2920RS001A01F01.FP_PARAM.AlarmDelay_L1_Acc" : Int AT %DB5048.DBW126, 500 ms
   "2920RS001A01F01.FP_PARAM.AlarmDelay_L2_Pre" : Int AT %DB5048.DBW128, 500 ms
   "2920RS001A01F01.FP_PARAM.AlarmDelay_L2_Acc" : Int AT %DB5048.DBW130, 500 ms
   "2920RS001A01F01.FP_PARAM.AlarmDelay_L3_Pre" : Int AT %DB5048.DBW132, 500 ms
   "2920RS001A01F01.FP_PARAM.AlarmDelay_L3_Acc" : Int AT %DB5048.DBW134, 500 ms
   "2920RS001A01F01.FP_PARAM.OpenLoopDelay_Pre" : Int AT %DB5048.DBW136, 500 ms
   "2920RS001A01F01.FP_PARAM.OpenLoopDelay_Acc" : Int AT %DB5048.DBW138, 500 ms
   "2920RS001A01F01.FP_PARAM.OverRangeDelay_Pre" : Int AT %DB5048.DBW140, 500 ms
   "2920RS001A01F01.FP_PARAM.OverRangeDelay_Acc" : Int AT %DB5048.DBW142, 500 ms
   "2920RS001A01F01.FP_PARAM.AuxLimit_H2_Value" : Real AT %DB5048.DBD144, 500 ms
   "2920RS001A01F01.FP_PARAM.AuxLimit_H1_Value" : Real AT %DB5048.DBD148, 500 ms
   "2920RS001A01F01.FP_PARAM.AuxLimit_L2_Value" : Real AT %DB5048.DBD152, 500 ms
   "2920RS001A01F01.FP_PARAM.AuxLimit_L1_Value" : Real AT %DB5048.DBD156, 500 ms
   "2920RS001A01F01.Unit" : TextRef, internal   // Еденицы измерения При експорте из ECS через скрипт заполняется автоматически, если теги копируются в ручную то требуется задатать свойство Text
   "2920RS001A01F01.Decimals" : TextRef, internal   // Формат отображения При експорте из ECS через скрипт, заполняется автоматически. Если теги копируются в ручную то требуется задатать свойство Text s999999.9
   "2920RS001A01F01.FP_EN.Square" : Bool AT %DB5048.DBX46.0, 500 ms
   "2920RS001A01F01.FP_EN.SquareRoot" : Bool AT %DB5048.DBX46.1, 500 ms
   "2920RS001A01F01.FP_EN.ParentSupress" : Bool AT %DB5048.DBX46.2, 500 ms
   "2920RS001A01F01.FP_EN.ParentSupressUnit" : Bool AT %DB5048.DBX46.3, 500 ms
   "2920RS001A01F01.FP_EN.Force" : Bool AT %DB5048.DBX46.4, 500 ms
   "2920RS001A01F01.FP_EN.Damping" : Bool AT %DB5048.DBX46.5, 500 ms
   "2920RS001A01F01.FP_EN.Gradient_Pos" : Bool AT %DB5048.DBX46.6, 500 ms
   "2920RS001A01F01.FP_EN.Gradient_Neg" : Bool AT %DB5048.DBX46.7, 500 ms
   "2920RS001A01F01.FP_EN.Hysteresis" : Bool AT %DB5048.DBX47.0, 500 ms
   "2920RS001A01F01.FP_EN.Alarm_H3" : Bool AT %DB5048.DBX47.1, 500 ms
   "2920RS001A01F01.FP_EN.Alarm_H2" : Bool AT %DB5048.DBX47.2, 500 ms
   "2920RS001A01F01.FP_EN.Alarm_H1" : Bool AT %DB5048.DBX47.3, 500 ms
   "2920RS001A01F01.FP_EN.Alarm_L1" : Bool AT %DB5048.DBX47.4, 500 ms
   "2920RS001A01F01.FP_EN.Alarm_L2" : Bool AT %DB5048.DBX47.5, 500 ms
   "2920RS001A01F01.FP_EN.Alarm_L3" : Bool AT %DB5048.DBX47.6, 500 ms
   "2920RS001A01F01.FP_EN.AlarmDelay_H3" : Bool AT %DB5048.DBX47.7, 500 ms
   "2920RS001A01F01.FP_EN.AlarmDelay_H2" : Bool AT %DB5048.DBX48.0, 500 ms
   "2920RS001A01F01.FP_EN.AlarmDelay_H1" : Bool AT %DB5048.DBX48.1, 500 ms
   "2920RS001A01F01.FP_EN.AlarmDelay_L1" : Bool AT %DB5048.DBX48.2, 500 ms
   "2920RS001A01F01.FP_EN.AlarmDelay_L2" : Bool AT %DB5048.DBX48.3, 500 ms
   "2920RS001A01F01.FP_EN.AlarmDelay_L3" : Bool AT %DB5048.DBX48.4, 500 ms
   "2920RS001A01F01.FP_EN.ROC_Warn" : Bool AT %DB5048.DBX48.5, 500 ms
   "2920RS001A01F01.FP_EN.U_Range_Warn" : Bool AT %DB5048.DBX48.6, 500 ms
   "2920RS001A01F01.FP_EN.O_Range_Warn" : Bool AT %DB5048.DBX48.7, 500 ms
   "2920RS001A01F01.trend_tag_name" : TextRef, internal   // Еденицы измерения При експорте из ECS через скрипт - заполняется автоматически, если теги копируются в ручную то требуется задатать свойство Text - имя тега для тренда
   "2920RS001A01F01.DQ.AL_H3" : Bool AT %DB5048.DBX16.0, 500 ms
   "2920RS001A01F01.DQ.AL_H2" : Bool AT %DB5048.DBX16.1, 500 ms
   "2920RS001A01F01.DQ.AL_H1" : Bool AT %DB5048.DBX16.2, 500 ms
   "2920RS001A01F01.DQ.AL_L1" : Bool AT %DB5048.DBX16.3, 500 ms
   "2920RS001A01F01.DQ.AL_L2" : Bool AT %DB5048.DBX16.4, 500 ms
   "2920RS001A01F01.DQ.AL_L3" : Bool AT %DB5048.DBX16.5, 500 ms
   "2920RS001A01F01.DQ.SIG_OK" : Bool AT %DB5048.DBX16.6, 500 ms
   "2920RS001A01F01.DQ.LIM_H2" : Bool AT %DB5048.DBX16.7, 500 ms
   "2920RS001A01F01.DQ.LIM_H1" : Bool AT %DB5048.DBX17.0, 500 ms
   "2920RS001A01F01.DQ.LIM_L1" : Bool AT %DB5048.DBX17.1, 500 ms
   "2920RS001A01F01.DQ.LIM_L2" : Bool AT %DB5048.DBX17.2, 500 ms
   "2920RS001A01F01.DQ.GR_P" : Bool AT %DB5048.DBX17.3, 500 ms
   "2920RS001A01F01.DQ.GR_N" : Bool AT %DB5048.DBX17.4, 500 ms
   "2920RS001A01F01.I.IN" : Real AT %DB5048.DBD2, 500 ms
   "2920RS001A01F01.I.SIG_TYPE" : Int AT %DB5048.DBW0, 500 ms
   "2920RS001A01F01.I.FI_BUS" : Byte AT %DB5048.DBB6, 500 ms
   "2920RS001A01F01.DI.U_RANGE" : Bool AT %DB5048.DBX7.0, 500 ms
   "2920RS001A01F01.DI.O_RANGE" : Bool AT %DB5048.DBX7.1, 500 ms
   "2920RS001A01F01.DI.SIG_FAULT" : Bool AT %DB5048.DBX7.2, 500 ms
   "2920RS001A01F01.DI.EnConfig" : Bool AT %DB5048.DBX7.3, 500 ms
   "2920RS001A01F01.DI.AEN" : Bool AT %DB5048.DBX7.4, 500 ms
   "2920RS001A01F01.DI.AL_SUPR" : Bool AT %DB5048.DBX7.5, 500 ms
   "2920RS001A01F01.Q.PV_NORM" : Real AT %DB5048.DBD8, 500 ms
   "2920RS001A01F01.Q.PV_SCAL" : Real AT %DB5048.DBD12, 500 ms
   "2920RS001A01F01.ParentInfo" : TextRef, internal   // Имя родителя для попап окна, вкладка инфо. При експорте из ECS через скрипт заполняется автоматически, если теги копируются в ручную то требуется в ручную задатать свойство Start Value

HMI tags "2920RS001A01F02"
   "2920RS001A01F02.MSW" : 52809b66-421d-457f-8884-6f7a49d4e247 AT %DB5049.DBX18.0, 500 ms
   "2920RS001A01F02.DefaultText" : TextRef, internal   // Заголовок POPUP окна. При експорте из ECS через скрипт заполняется автоматически, если теги копируются в ручную то требуется в ручную задатать свойство Start Value
   "2920RS001A01F02.BlockInfo" : Array [0..2] of Int AT %DB5049.DBX38.0, 500 ms
   "2920RS001A01F02.StatusWork" : Int AT %DB5049.DBW242, 500 ms
   "2920RS001A01F02.FP_PARAM.DampingTime" : Int AT %DB5049.DBW50, 500 ms
   "2920RS001A01F02.FP_PARAM.Force_Value" : Real AT %DB5049.DBD52, 500 ms
   "2920RS001A01F02.FP_PARAM.Scale_Min" : Real AT %DB5049.DBD56, 500 ms
   "2920RS001A01F02.FP_PARAM.Scale_Max" : Real AT %DB5049.DBD60, 500 ms
   "2920RS001A01F02.FP_PARAM.Gradient" : Real AT %DB5049.DBD64, 500 ms
   "2920RS001A01F02.FP_PARAM.Grad_Pos" : Real AT %DB5049.DBD68, 500 ms
   "2920RS001A01F02.FP_PARAM.Grad_Neg" : Real AT %DB5049.DBD72, 500 ms
   "2920RS001A01F02.FP_PARAM.Grad_X" : Real AT %DB5049.DBD76, 500 ms
   "2920RS001A01F02.FP_PARAM.Gradient_Time_Pre" : Int AT %DB5049.DBW80, 500 ms
   "2920RS001A01F02.FP_PARAM.Gradient_Time_ACC" : Int AT %DB5049.DBW82, 500 ms
   "2920RS001A01F02.FP_PARAM.Alarm_Hyst" : Real AT %DB5049.DBD84, 500 ms
   "2920RS001A01F02.FP_PARAM.AlarmLimit_H3" : Real AT %DB5049.DBD88, 500 ms
   "2920RS001A01F02.FP_PARAM.AlarmLimit_H2" : Real AT %DB5049.DBD92, 500 ms
   "2920RS001A01F02.FP_PARAM.AlarmLimit_H1" : Real AT %DB5049.DBD96, 500 ms
   "2920RS001A01F02.FP_PARAM.AlarmLimit_L1" : Real AT %DB5049.DBD100, 500 ms
   "2920RS001A01F02.FP_PARAM.AlarmLimit_L2" : Real AT %DB5049.DBD104, 500 ms
   "2920RS001A01F02.FP_PARAM.AlarmLimit_L3" : Real AT %DB5049.DBD108, 500 ms
   "2920RS001A01F02.FP_PARAM.AlarmDelay_H3_Pre" : Int AT %DB5049.DBW112, 500 ms
   "2920RS001A01F02.FP_PARAM.AlarmDelay_H3_Acc" : Int AT %DB5049.DBW114, 500 ms
   "2920RS001A01F02.FP_PARAM.AlarmDelay_H2_Pre" : Int AT %DB5049.DBW116, 500 ms
   "2920RS001A01F02.FP_PARAM.AlarmDelay_H2_Acc" : Int AT %DB5049.DBW118, 500 ms
   "2920RS001A01F02.FP_PARAM.AlarmDelay_H1_Pre" : Int AT %DB5049.DBW120, 500 ms
   "2920RS001A01F02.FP_PARAM.AlarmDelay_H1_Acc" : Int AT %DB5049.DBW122, 500 ms
   "2920RS001A01F02.FP_PARAM.AlarmDelay_L1_Pre" : Int AT %DB5049.DBW124, 500 ms
   "2920RS001A01F02.FP_PARAM.AlarmDelay_L1_Acc" : Int AT %DB5049.DBW126, 500 ms
   "2920RS001A01F02.FP_PARAM.AlarmDelay_L2_Pre" : Int AT %DB5049.DBW128, 500 ms
   "2920RS001A01F02.FP_PARAM.AlarmDelay_L2_Acc" : Int AT %DB5049.DBW130, 500 ms
   "2920RS001A01F02.FP_PARAM.AlarmDelay_L3_Pre" : Int AT %DB5049.DBW132, 500 ms
   "2920RS001A01F02.FP_PARAM.AlarmDelay_L3_Acc" : Int AT %DB5049.DBW134, 500 ms
   "2920RS001A01F02.FP_PARAM.OpenLoopDelay_Pre" : Int AT %DB5049.DBW136, 500 ms
   "2920RS001A01F02.FP_PARAM.OpenLoopDelay_Acc" : Int AT %DB5049.DBW138, 500 ms
   "2920RS001A01F02.FP_PARAM.OverRangeDelay_Pre" : Int AT %DB5049.DBW140, 500 ms
   "2920RS001A01F02.FP_PARAM.OverRangeDelay_Acc" : Int AT %DB5049.DBW142, 500 ms
   "2920RS001A01F02.FP_PARAM.AuxLimit_H2_Value" : Real AT %DB5049.DBD144, 500 ms
   "2920RS001A01F02.FP_PARAM.AuxLimit_H1_Value" : Real AT %DB5049.DBD148, 500 ms
   "2920RS001A01F02.FP_PARAM.AuxLimit_L2_Value" : Real AT %DB5049.DBD152, 500 ms
   "2920RS001A01F02.FP_PARAM.AuxLimit_L1_Value" : Real AT %DB5049.DBD156, 500 ms
   "2920RS001A01F02.Unit" : TextRef, internal   // Еденицы измерения При експорте из ECS через скрипт заполняется автоматически, если теги копируются в ручную то требуется задатать свойство Text
   "2920RS001A01F02.Decimals" : TextRef, internal   // Формат отображения При експорте из ECS через скрипт, заполняется автоматически. Если теги копируются в ручную то требуется задатать свойство Text s999999.9
   "2920RS001A01F02.FP_EN.Square" : Bool AT %DB5049.DBX46.0, 500 ms
   "2920RS001A01F02.FP_EN.SquareRoot" : Bool AT %DB5049.DBX46.1, 500 ms
   "2920RS001A01F02.FP_EN.ParentSupress" : Bool AT %DB5049.DBX46.2, 500 ms
   "2920RS001A01F02.FP_EN.ParentSupressUnit" : Bool AT %DB5049.DBX46.3, 500 ms
   "2920RS001A01F02.FP_EN.Force" : Bool AT %DB5049.DBX46.4, 500 ms
   "2920RS001A01F02.FP_EN.Damping" : Bool AT %DB5049.DBX46.5, 500 ms
   "2920RS001A01F02.FP_EN.Gradient_Pos" : Bool AT %DB5049.DBX46.6, 500 ms
   "2920RS001A01F02.FP_EN.Gradient_Neg" : Bool AT %DB5049.DBX46.7, 500 ms
   "2920RS001A01F02.FP_EN.Hysteresis" : Bool AT %DB5049.DBX47.0, 500 ms
   "2920RS001A01F02.FP_EN.Alarm_H3" : Bool AT %DB5049.DBX47.1, 500 ms
   "2920RS001A01F02.FP_EN.Alarm_H2" : Bool AT %DB5049.DBX47.2, 500 ms
   "2920RS001A01F02.FP_EN.Alarm_H1" : Bool AT %DB5049.DBX47.3, 500 ms
   "2920RS001A01F02.FP_EN.Alarm_L1" : Bool AT %DB5049.DBX47.4, 500 ms
   "2920RS001A01F02.FP_EN.Alarm_L2" : Bool AT %DB5049.DBX47.5, 500 ms
   "2920RS001A01F02.FP_EN.Alarm_L3" : Bool AT %DB5049.DBX47.6, 500 ms
   "2920RS001A01F02.FP_EN.AlarmDelay_H3" : Bool AT %DB5049.DBX47.7, 500 ms
   "2920RS001A01F02.FP_EN.AlarmDelay_H2" : Bool AT %DB5049.DBX48.0, 500 ms
   "2920RS001A01F02.FP_EN.AlarmDelay_H1" : Bool AT %DB5049.DBX48.1, 500 ms
   "2920RS001A01F02.FP_EN.AlarmDelay_L1" : Bool AT %DB5049.DBX48.2, 500 ms
   "2920RS001A01F02.FP_EN.AlarmDelay_L2" : Bool AT %DB5049.DBX48.3, 500 ms
   "2920RS001A01F02.FP_EN.AlarmDelay_L3" : Bool AT %DB5049.DBX48.4, 500 ms
   "2920RS001A01F02.FP_EN.ROC_Warn" : Bool AT %DB5049.DBX48.5, 500 ms
   "2920RS001A01F02.FP_EN.U_Range_Warn" : Bool AT %DB5049.DBX48.6, 500 ms
   "2920RS001A01F02.FP_EN.O_Range_Warn" : Bool AT %DB5049.DBX48.7, 500 ms
   "2920RS001A01F02.trend_tag_name" : TextRef, internal   // Еденицы измерения При експорте из ECS через скрипт - заполняется автоматически, если теги копируются в ручную то требуется задатать свойство Text - имя тега для тренда
   "2920RS001A01F02.DQ.AL_H3" : Bool AT %DB5049.DBX16.0, 500 ms
   "2920RS001A01F02.DQ.AL_H2" : Bool AT %DB5049.DBX16.1, 500 ms
   "2920RS001A01F02.DQ.AL_H1" : Bool AT %DB5049.DBX16.2, 500 ms
   "2920RS001A01F02.DQ.AL_L1" : Bool AT %DB5049.DBX16.3, 500 ms
   "2920RS001A01F02.DQ.AL_L2" : Bool AT %DB5049.DBX16.4, 500 ms
   "2920RS001A01F02.DQ.AL_L3" : Bool AT %DB5049.DBX16.5, 500 ms
   "2920RS001A01F02.DQ.SIG_OK" : Bool AT %DB5049.DBX16.6, 500 ms
   "2920RS001A01F02.DQ.LIM_H2" : Bool AT %DB5049.DBX16.7, 500 ms
   "2920RS001A01F02.DQ.LIM_H1" : Bool AT %DB5049.DBX17.0, 500 ms
   "2920RS001A01F02.DQ.LIM_L1" : Bool AT %DB5049.DBX17.1, 500 ms
   "2920RS001A01F02.DQ.LIM_L2" : Bool AT %DB5049.DBX17.2, 500 ms
   "2920RS001A01F02.DQ.GR_P" : Bool AT %DB5049.DBX17.3, 500 ms
   "2920RS001A01F02.DQ.GR_N" : Bool AT %DB5049.DBX17.4, 500 ms
   "2920RS001A01F02.I.IN" : Real AT %DB5049.DBD2, 500 ms
   "2920RS001A01F02.I.SIG_TYPE" : Int AT %DB5049.DBW0, 500 ms
   "2920RS001A01F02.I.FI_BUS" : Byte AT %DB5049.DBB6, 500 ms
   "2920RS001A01F02.DI.U_RANGE" : Bool AT %DB5049.DBX7.0, 500 ms
   "2920RS001A01F02.DI.O_RANGE" : Bool AT %DB5049.DBX7.1, 500 ms
   "2920RS001A01F02.DI.SIG_FAULT" : Bool AT %DB5049.DBX7.2, 500 ms
   "2920RS001A01F02.DI.EnConfig" : Bool AT %DB5049.DBX7.3, 500 ms
   "2920RS001A01F02.DI.AEN" : Bool AT %DB5049.DBX7.4, 500 ms
   "2920RS001A01F02.DI.AL_SUPR" : Bool AT %DB5049.DBX7.5, 500 ms
   "2920RS001A01F02.Q.PV_NORM" : Real AT %DB5049.DBD8, 500 ms
   "2920RS001A01F02.Q.PV_SCAL" : Real AT %DB5049.DBD12, 500 ms
   "2920RS001A01F02.ParentInfo" : TextRef, internal   // Имя родителя для попап окна, вкладка инфо. При експорте из ECS через скрипт заполняется автоматически, если теги копируются в ручную то требуется в ручную задатать свойство Start Value

HMI tags "2920RS001A01L01"
   "2920RS001A01L01.MSW" : 52809b66-421d-457f-8884-6f7a49d4e247 AT %DB5050.DBX18.0, 500 ms
   "2920RS001A01L01.DefaultText" : TextRef, internal   // Заголовок POPUP окна. При експорте из ECS через скрипт заполняется автоматически, если теги копируются в ручную то требуется в ручную задатать свойство Start Value
   "2920RS001A01L01.BlockInfo" : Array [0..2] of Int AT %DB5050.DBX38.0, 500 ms
   "2920RS001A01L01.StatusWork" : Int AT %DB5050.DBW242, 500 ms
   "2920RS001A01L01.FP_PARAM.DampingTime" : Int AT %DB5050.DBW50, 500 ms
   "2920RS001A01L01.FP_PARAM.Force_Value" : Real AT %DB5050.DBD52, 500 ms
   "2920RS001A01L01.FP_PARAM.Scale_Min" : Real AT %DB5050.DBD56, 500 ms
   "2920RS001A01L01.FP_PARAM.Scale_Max" : Real AT %DB5050.DBD60, 500 ms
   "2920RS001A01L01.FP_PARAM.Gradient" : Real AT %DB5050.DBD64, 500 ms
   "2920RS001A01L01.FP_PARAM.Grad_Pos" : Real AT %DB5050.DBD68, 500 ms
   "2920RS001A01L01.FP_PARAM.Grad_Neg" : Real AT %DB5050.DBD72, 500 ms
   "2920RS001A01L01.FP_PARAM.Grad_X" : Real AT %DB5050.DBD76, 500 ms
   "2920RS001A01L01.FP_PARAM.Gradient_Time_Pre" : Int AT %DB5050.DBW80, 500 ms
   "2920RS001A01L01.FP_PARAM.Gradient_Time_ACC" : Int AT %DB5050.DBW82, 500 ms
   "2920RS001A01L01.FP_PARAM.Alarm_Hyst" : Real AT %DB5050.DBD84, 500 ms
   "2920RS001A01L01.FP_PARAM.AlarmLimit_H3" : Real AT %DB5050.DBD88, 500 ms
   "2920RS001A01L01.FP_PARAM.AlarmLimit_H2" : Real AT %DB5050.DBD92, 500 ms
   "2920RS001A01L01.FP_PARAM.AlarmLimit_H1" : Real AT %DB5050.DBD96, 500 ms
   "2920RS001A01L01.FP_PARAM.AlarmLimit_L1" : Real AT %DB5050.DBD100, 500 ms
   "2920RS001A01L01.FP_PARAM.AlarmLimit_L2" : Real AT %DB5050.DBD104, 500 ms
   "2920RS001A01L01.FP_PARAM.AlarmLimit_L3" : Real AT %DB5050.DBD108, 500 ms
   "2920RS001A01L01.FP_PARAM.AlarmDelay_H3_Pre" : Int AT %DB5050.DBW112, 500 ms
   "2920RS001A01L01.FP_PARAM.AlarmDelay_H3_Acc" : Int AT %DB5050.DBW114, 500 ms
   "2920RS001A01L01.FP_PARAM.AlarmDelay_H2_Pre" : Int AT %DB5050.DBW116, 500 ms
   "2920RS001A01L01.FP_PARAM.AlarmDelay_H2_Acc" : Int AT %DB5050.DBW118, 500 ms
   "2920RS001A01L01.FP_PARAM.AlarmDelay_H1_Pre" : Int AT %DB5050.DBW120, 500 ms
   "2920RS001A01L01.FP_PARAM.AlarmDelay_H1_Acc" : Int AT %DB5050.DBW122, 500 ms
   "2920RS001A01L01.FP_PARAM.AlarmDelay_L1_Pre" : Int AT %DB5050.DBW124, 500 ms
   "2920RS001A01L01.FP_PARAM.AlarmDelay_L1_Acc" : Int AT %DB5050.DBW126, 500 ms
   "2920RS001A01L01.FP_PARAM.AlarmDelay_L2_Pre" : Int AT %DB5050.DBW128, 500 ms
   "2920RS001A01L01.FP_PARAM.AlarmDelay_L2_Acc" : Int AT %DB5050.DBW130, 500 ms
   "2920RS001A01L01.FP_PARAM.AlarmDelay_L3_Pre" : Int AT %DB5050.DBW132, 500 ms
   "2920RS001A01L01.FP_PARAM.AlarmDelay_L3_Acc" : Int AT %DB5050.DBW134, 500 ms
   "2920RS001A01L01.FP_PARAM.OpenLoopDelay_Pre" : Int AT %DB5050.DBW136, 500 ms
   "2920RS001A01L01.FP_PARAM.OpenLoopDelay_Acc" : Int AT %DB5050.DBW138, 500 ms
   "2920RS001A01L01.FP_PARAM.OverRangeDelay_Pre" : Int AT %DB5050.DBW140, 500 ms
   "2920RS001A01L01.FP_PARAM.OverRangeDelay_Acc" : Int AT %DB5050.DBW142, 500 ms
   "2920RS001A01L01.FP_PARAM.AuxLimit_H2_Value" : Real AT %DB5050.DBD144, 500 ms
   "2920RS001A01L01.FP_PARAM.AuxLimit_H1_Value" : Real AT %DB5050.DBD148, 500 ms
   "2920RS001A01L01.FP_PARAM.AuxLimit_L2_Value" : Real AT %DB5050.DBD152, 500 ms
   "2920RS001A01L01.FP_PARAM.AuxLimit_L1_Value" : Real AT %DB5050.DBD156, 500 ms
   "2920RS001A01L01.Unit" : TextRef, internal   // Еденицы измерения При експорте из ECS через скрипт заполняется автоматически, если теги копируются в ручную то требуется задатать свойство Text
   "2920RS001A01L01.Decimals" : TextRef, internal   // Формат отображения При експорте из ECS через скрипт, заполняется автоматически. Если теги копируются в ручную то требуется задатать свойство Text s999999.9
   "2920RS001A01L01.FP_EN.Square" : Bool AT %DB5050.DBX46.0, 500 ms
   "2920RS001A01L01.FP_EN.SquareRoot" : Bool AT %DB5050.DBX46.1, 500 ms
   "2920RS001A01L01.FP_EN.ParentSupress" : Bool AT %DB5050.DBX46.2, 500 ms
   "2920RS001A01L01.FP_EN.ParentSupressUnit" : Bool AT %DB5050.DBX46.3, 500 ms
   "2920RS001A01L01.FP_EN.Force" : Bool AT %DB5050.DBX46.4, 500 ms
   "2920RS001A01L01.FP_EN.Damping" : Bool AT %DB5050.DBX46.5, 500 ms
   "2920RS001A01L01.FP_EN.Gradient_Pos" : Bool AT %DB5050.DBX46.6, 500 ms
   "2920RS001A01L01.FP_EN.Gradient_Neg" : Bool AT %DB5050.DBX46.7, 500 ms
   "2920RS001A01L01.FP_EN.Hysteresis" : Bool AT %DB5050.DBX47.0, 500 ms
   "2920RS001A01L01.FP_EN.Alarm_H3" : Bool AT %DB5050.DBX47.1, 500 ms
   "2920RS001A01L01.FP_EN.Alarm_H2" : Bool AT %DB5050.DBX47.2, 500 ms
   "2920RS001A01L01.FP_EN.Alarm_H1" : Bool AT %DB5050.DBX47.3, 500 ms
   "2920RS001A01L01.FP_EN.Alarm_L1" : Bool AT %DB5050.DBX47.4, 500 ms
   "2920RS001A01L01.FP_EN.Alarm_L2" : Bool AT %DB5050.DBX47.5, 500 ms
   "2920RS001A01L01.FP_EN.Alarm_L3" : Bool AT %DB5050.DBX47.6, 500 ms
   "2920RS001A01L01.FP_EN.AlarmDelay_H3" : Bool AT %DB5050.DBX47.7, 500 ms
   "2920RS001A01L01.FP_EN.AlarmDelay_H2" : Bool AT %DB5050.DBX48.0, 500 ms
   "2920RS001A01L01.FP_EN.AlarmDelay_H1" : Bool AT %DB5050.DBX48.1, 500 ms
   "2920RS001A01L01.FP_EN.AlarmDelay_L1" : Bool AT %DB5050.DBX48.2, 500 ms
   "2920RS001A01L01.FP_EN.AlarmDelay_L2" : Bool AT %DB5050.DBX48.3, 500 ms
   "2920RS001A01L01.FP_EN.AlarmDelay_L3" : Bool AT %DB5050.DBX48.4, 500 ms
   "2920RS001A01L01.FP_EN.ROC_Warn" : Bool AT %DB5050.DBX48.5, 500 ms
   "2920RS001A01L01.FP_EN.U_Range_Warn" : Bool AT %DB5050.DBX48.6, 500 ms
   "2920RS001A01L01.FP_EN.O_Range_Warn" : Bool AT %DB5050.DBX48.7, 500 ms
   "2920RS001A01L01.trend_tag_name" : TextRef, internal   // Еденицы измерения При експорте из ECS через скрипт - заполняется автоматически, если теги копируются в ручную то требуется задатать свойство Text - имя тега для тренда
   "2920RS001A01L01.DQ.AL_H3" : Bool AT %DB5050.DBX16.0, 500 ms
   "2920RS001A01L01.DQ.AL_H2" : Bool AT %DB5050.DBX16.1, 500 ms
   "2920RS001A01L01.DQ.AL_H1" : Bool AT %DB5050.DBX16.2, 500 ms
   "2920RS001A01L01.DQ.AL_L1" : Bool AT %DB5050.DBX16.3, 500 ms
   "2920RS001A01L01.DQ.AL_L2" : Bool AT %DB5050.DBX16.4, 500 ms
   "2920RS001A01L01.DQ.AL_L3" : Bool AT %DB5050.DBX16.5, 500 ms
   "2920RS001A01L01.DQ.SIG_OK" : Bool AT %DB5050.DBX16.6, 500 ms
   "2920RS001A01L01.DQ.LIM_H2" : Bool AT %DB5050.DBX16.7, 500 ms
   "2920RS001A01L01.DQ.LIM_H1" : Bool AT %DB5050.DBX17.0, 500 ms
   "2920RS001A01L01.DQ.LIM_L1" : Bool AT %DB5050.DBX17.1, 500 ms
   "2920RS001A01L01.DQ.LIM_L2" : Bool AT %DB5050.DBX17.2, 500 ms
   "2920RS001A01L01.DQ.GR_P" : Bool AT %DB5050.DBX17.3, 500 ms
   "2920RS001A01L01.DQ.GR_N" : Bool AT %DB5050.DBX17.4, 500 ms
   "2920RS001A01L01.I.IN" : Real AT %DB5050.DBD2, 500 ms
   "2920RS001A01L01.I.SIG_TYPE" : Int AT %DB5050.DBW0, 500 ms
   "2920RS001A01L01.I.FI_BUS" : Byte AT %DB5050.DBB6, 500 ms
   "2920RS001A01L01.DI.U_RANGE" : Bool AT %DB5050.DBX7.0, 500 ms
   "2920RS001A01L01.DI.O_RANGE" : Bool AT %DB5050.DBX7.1, 500 ms
   "2920RS001A01L01.DI.SIG_FAULT" : Bool AT %DB5050.DBX7.2, 500 ms
   "2920RS001A01L01.DI.EnConfig" : Bool AT %DB5050.DBX7.3, 500 ms
   "2920RS001A01L01.DI.AEN" : Bool AT %DB5050.DBX7.4, 500 ms
   "2920RS001A01L01.DI.AL_SUPR" : Bool AT %DB5050.DBX7.5, 500 ms
   "2920RS001A01L01.Q.PV_NORM" : Real AT %DB5050.DBD8, 500 ms
   "2920RS001A01L01.Q.PV_SCAL" : Real AT %DB5050.DBD12, 500 ms
   "2920RS001A01L01.ParentInfo" : TextRef, internal   // Имя родителя для попап окна, вкладка инфо. При експорте из ECS через скрипт заполняется автоматически, если теги копируются в ручную то требуется в ручную задатать свойство Start Value

HMI tags "2920RS001A01L02"
   "2920RS001A01L02.MSW" : 52809b66-421d-457f-8884-6f7a49d4e247 AT %DB5051.DBX18.0, 500 ms
   "2920RS001A01L02.DefaultText" : TextRef, internal   // Заголовок POPUP окна. При експорте из ECS через скрипт заполняется автоматически, если теги копируются в ручную то требуется в ручную задатать свойство Start Value
   "2920RS001A01L02.BlockInfo" : Array [0..2] of Int AT %DB5051.DBX38.0, 500 ms
   "2920RS001A01L02.StatusWork" : Int AT %DB5051.DBW242, 500 ms
   "2920RS001A01L02.FP_PARAM.DampingTime" : Int AT %DB5051.DBW50, 500 ms
   "2920RS001A01L02.FP_PARAM.Force_Value" : Real AT %DB5051.DBD52, 500 ms
   "2920RS001A01L02.FP_PARAM.Scale_Min" : Real AT %DB5051.DBD56, 500 ms
   "2920RS001A01L02.FP_PARAM.Scale_Max" : Real AT %DB5051.DBD60, 500 ms
   "2920RS001A01L02.FP_PARAM.Gradient" : Real AT %DB5051.DBD64, 500 ms
   "2920RS001A01L02.FP_PARAM.Grad_Pos" : Real AT %DB5051.DBD68, 500 ms
   "2920RS001A01L02.FP_PARAM.Grad_Neg" : Real AT %DB5051.DBD72, 500 ms
   "2920RS001A01L02.FP_PARAM.Grad_X" : Real AT %DB5051.DBD76, 500 ms
   "2920RS001A01L02.FP_PARAM.Gradient_Time_Pre" : Int AT %DB5051.DBW80, 500 ms
   "2920RS001A01L02.FP_PARAM.Gradient_Time_ACC" : Int AT %DB5051.DBW82, 500 ms
   "2920RS001A01L02.FP_PARAM.Alarm_Hyst" : Real AT %DB5051.DBD84, 500 ms
   "2920RS001A01L02.FP_PARAM.AlarmLimit_H3" : Real AT %DB5051.DBD88, 500 ms
   "2920RS001A01L02.FP_PARAM.AlarmLimit_H2" : Real AT %DB5051.DBD92, 500 ms
   "2920RS001A01L02.FP_PARAM.AlarmLimit_H1" : Real AT %DB5051.DBD96, 500 ms
   "2920RS001A01L02.FP_PARAM.AlarmLimit_L1" : Real AT %DB5051.DBD100, 500 ms
   "2920RS001A01L02.FP_PARAM.AlarmLimit_L2" : Real AT %DB5051.DBD104, 500 ms
   "2920RS001A01L02.FP_PARAM.AlarmLimit_L3" : Real AT %DB5051.DBD108, 500 ms
   "2920RS001A01L02.FP_PARAM.AlarmDelay_H3_Pre" : Int AT %DB5051.DBW112, 500 ms
   "2920RS001A01L02.FP_PARAM.AlarmDelay_H3_Acc" : Int AT %DB5051.DBW114, 500 ms
   "2920RS001A01L02.FP_PARAM.AlarmDelay_H2_Pre" : Int AT %DB5051.DBW116, 500 ms
   "2920RS001A01L02.FP_PARAM.AlarmDelay_H2_Acc" : Int AT %DB5051.DBW118, 500 ms
   "2920RS001A01L02.FP_PARAM.AlarmDelay_H1_Pre" : Int AT %DB5051.DBW120, 500 ms
   "2920RS001A01L02.FP_PARAM.AlarmDelay_H1_Acc" : Int AT %DB5051.DBW122, 500 ms
   "2920RS001A01L02.FP_PARAM.AlarmDelay_L1_Pre" : Int AT %DB5051.DBW124, 500 ms
   "2920RS001A01L02.FP_PARAM.AlarmDelay_L1_Acc" : Int AT %DB5051.DBW126, 500 ms
   "2920RS001A01L02.FP_PARAM.AlarmDelay_L2_Pre" : Int AT %DB5051.DBW128, 500 ms
   "2920RS001A01L02.FP_PARAM.AlarmDelay_L2_Acc" : Int AT %DB5051.DBW130, 500 ms
   "2920RS001A01L02.FP_PARAM.AlarmDelay_L3_Pre" : Int AT %DB5051.DBW132, 500 ms
   "2920RS001A01L02.FP_PARAM.AlarmDelay_L3_Acc" : Int AT %DB5051.DBW134, 500 ms
   "2920RS001A01L02.FP_PARAM.OpenLoopDelay_Pre" : Int AT %DB5051.DBW136, 500 ms
   "2920RS001A01L02.FP_PARAM.OpenLoopDelay_Acc" : Int AT %DB5051.DBW138, 500 ms
   "2920RS001A01L02.FP_PARAM.OverRangeDelay_Pre" : Int AT %DB5051.DBW140, 500 ms
   "2920RS001A01L02.FP_PARAM.OverRangeDelay_Acc" : Int AT %DB5051.DBW142, 500 ms
   "2920RS001A01L02.FP_PARAM.AuxLimit_H2_Value" : Real AT %DB5051.DBD144, 500 ms
   "2920RS001A01L02.FP_PARAM.AuxLimit_H1_Value" : Real AT %DB5051.DBD148, 500 ms
   "2920RS001A01L02.FP_PARAM.AuxLimit_L2_Value" : Real AT %DB5051.DBD152, 500 ms
   "2920RS001A01L02.FP_PARAM.AuxLimit_L1_Value" : Real AT %DB5051.DBD156, 500 ms
   "2920RS001A01L02.Unit" : TextRef, internal   // Еденицы измерения При експорте из ECS через скрипт заполняется автоматически, если теги копируются в ручную то требуется задатать свойство Text
   "2920RS001A01L02.Decimals" : TextRef, internal   // Формат отображения При експорте из ECS через скрипт, заполняется автоматически. Если теги копируются в ручную то требуется задатать свойство Text s999999.9
   "2920RS001A01L02.FP_EN.Square" : Bool AT %DB5051.DBX46.0, 500 ms
   "2920RS001A01L02.FP_EN.SquareRoot" : Bool AT %DB5051.DBX46.1, 500 ms
   "2920RS001A01L02.FP_EN.ParentSupress" : Bool AT %DB5051.DBX46.2, 500 ms
   "2920RS001A01L02.FP_EN.ParentSupressUnit" : Bool AT %DB5051.DBX46.3, 500 ms
   "2920RS001A01L02.FP_EN.Force" : Bool AT %DB5051.DBX46.4, 500 ms
   "2920RS001A01L02.FP_EN.Damping" : Bool AT %DB5051.DBX46.5, 500 ms
   "2920RS001A01L02.FP_EN.Gradient_Pos" : Bool AT %DB5051.DBX46.6, 500 ms
   "2920RS001A01L02.FP_EN.Gradient_Neg" : Bool AT %DB5051.DBX46.7, 500 ms
   "2920RS001A01L02.FP_EN.Hysteresis" : Bool AT %DB5051.DBX47.0, 500 ms
   "2920RS001A01L02.FP_EN.Alarm_H3" : Bool AT %DB5051.DBX47.1, 500 ms
   "2920RS001A01L02.FP_EN.Alarm_H2" : Bool AT %DB5051.DBX47.2, 500 ms
   "2920RS001A01L02.FP_EN.Alarm_H1" : Bool AT %DB5051.DBX47.3, 500 ms
   "2920RS001A01L02.FP_EN.Alarm_L1" : Bool AT %DB5051.DBX47.4, 500 ms
   "2920RS001A01L02.FP_EN.Alarm_L2" : Bool AT %DB5051.DBX47.5, 500 ms
   "2920RS001A01L02.FP_EN.Alarm_L3" : Bool AT %DB5051.DBX47.6, 500 ms
   "2920RS001A01L02.FP_EN.AlarmDelay_H3" : Bool AT %DB5051.DBX47.7, 500 ms
   "2920RS001A01L02.FP_EN.AlarmDelay_H2" : Bool AT %DB5051.DBX48.0, 500 ms
   "2920RS001A01L02.FP_EN.AlarmDelay_H1" : Bool AT %DB5051.DBX48.1, 500 ms
   "2920RS001A01L02.FP_EN.AlarmDelay_L1" : Bool AT %DB5051.DBX48.2, 500 ms
   "2920RS001A01L02.FP_EN.AlarmDelay_L2" : Bool AT %DB5051.DBX48.3, 500 ms
   "2920RS001A01L02.FP_EN.AlarmDelay_L3" : Bool AT %DB5051.DBX48.4, 500 ms
   "2920RS001A01L02.FP_EN.ROC_Warn" : Bool AT %DB5051.DBX48.5, 500 ms
   "2920RS001A01L02.FP_EN.U_Range_Warn" : Bool AT %DB5051.DBX48.6, 500 ms
   "2920RS001A01L02.FP_EN.O_Range_Warn" : Bool AT %DB5051.DBX48.7, 500 ms
   "2920RS001A01L02.trend_tag_name" : TextRef, internal   // Еденицы измерения При експорте из ECS через скрипт - заполняется автоматически, если теги копируются в ручную то требуется задатать свойство Text - имя тега для тренда
   "2920RS001A01L02.DQ.AL_H3" : Bool AT %DB5051.DBX16.0, 500 ms
   "2920RS001A01L02.DQ.AL_H2" : Bool AT %DB5051.DBX16.1, 500 ms
   "2920RS001A01L02.DQ.AL_H1" : Bool AT %DB5051.DBX16.2, 500 ms
   "2920RS001A01L02.DQ.AL_L1" : Bool AT %DB5051.DBX16.3, 500 ms
   "2920RS001A01L02.DQ.AL_L2" : Bool AT %DB5051.DBX16.4, 500 ms
   "2920RS001A01L02.DQ.AL_L3" : Bool AT %DB5051.DBX16.5, 500 ms
   "2920RS001A01L02.DQ.SIG_OK" : Bool AT %DB5051.DBX16.6, 500 ms
   "2920RS001A01L02.DQ.LIM_H2" : Bool AT %DB5051.DBX16.7, 500 ms
   "2920RS001A01L02.DQ.LIM_H1" : Bool AT %DB5051.DBX17.0, 500 ms
   "2920RS001A01L02.DQ.LIM_L1" : Bool AT %DB5051.DBX17.1, 500 ms
   "2920RS001A01L02.DQ.LIM_L2" : Bool AT %DB5051.DBX17.2, 500 ms
   "2920RS001A01L02.DQ.GR_P" : Bool AT %DB5051.DBX17.3, 500 ms
   "2920RS001A01L02.DQ.GR_N" : Bool AT %DB5051.DBX17.4, 500 ms
   "2920RS001A01L02.I.IN" : Real AT %DB5051.DBD2, 500 ms
   "2920RS001A01L02.I.SIG_TYPE" : Int AT %DB5051.DBW0, 500 ms
   "2920RS001A01L02.I.FI_BUS" : Byte AT %DB5051.DBB6, 500 ms
   "2920RS001A01L02.DI.U_RANGE" : Bool AT %DB5051.DBX7.0, 500 ms
   "2920RS001A01L02.DI.O_RANGE" : Bool AT %DB5051.DBX7.1, 500 ms
   "2920RS001A01L02.DI.SIG_FAULT" : Bool AT %DB5051.DBX7.2, 500 ms
   "2920RS001A01L02.DI.EnConfig" : Bool AT %DB5051.DBX7.3, 500 ms
   "2920RS001A01L02.DI.AEN" : Bool AT %DB5051.DBX7.4, 500 ms
   "2920RS001A01L02.DI.AL_SUPR" : Bool AT %DB5051.DBX7.5, 500 ms
   "2920RS001A01L02.Q.PV_NORM" : Real AT %DB5051.DBD8, 500 ms
   "2920RS001A01L02.Q.PV_SCAL" : Real AT %DB5051.DBD12, 500 ms
   "2920RS001A01L02.ParentInfo" : TextRef, internal   // Имя родителя для попап окна, вкладка инфо. При експорте из ECS через скрипт заполняется автоматически, если теги копируются в ручную то требуется в ручную задатать свойство Start Value

HMI tags "2920RS001A01T01"
   "2920RS001A01T01.MSW" : 52809b66-421d-457f-8884-6f7a49d4e247 AT %DB5052.DBX18.0, 500 ms
   "2920RS001A01T01.DefaultText" : TextRef, internal   // Заголовок POPUP окна. При експорте из ECS через скрипт заполняется автоматически, если теги копируются в ручную то требуется в ручную задатать свойство Start Value
   "2920RS001A01T01.BlockInfo" : Array [0..2] of Int AT %DB5052.DBX38.0, 500 ms
   "2920RS001A01T01.StatusWork" : Int AT %DB5052.DBW242, 500 ms
   "2920RS001A01T01.FP_PARAM.DampingTime" : Int AT %DB5052.DBW50, 500 ms
   "2920RS001A01T01.FP_PARAM.Force_Value" : Real AT %DB5052.DBD52, 500 ms
   "2920RS001A01T01.FP_PARAM.Scale_Min" : Real AT %DB5052.DBD56, 500 ms
   "2920RS001A01T01.FP_PARAM.Scale_Max" : Real AT %DB5052.DBD60, 500 ms
   "2920RS001A01T01.FP_PARAM.Gradient" : Real AT %DB5052.DBD64, 500 ms
   "2920RS001A01T01.FP_PARAM.Grad_Pos" : Real AT %DB5052.DBD68, 500 ms
   "2920RS001A01T01.FP_PARAM.Grad_Neg" : Real AT %DB5052.DBD72, 500 ms
   "2920RS001A01T01.FP_PARAM.Grad_X" : Real AT %DB5052.DBD76, 500 ms
   "2920RS001A01T01.FP_PARAM.Gradient_Time_Pre" : Int AT %DB5052.DBW80, 500 ms
   "2920RS001A01T01.FP_PARAM.Gradient_Time_ACC" : Int AT %DB5052.DBW82, 500 ms
   "2920RS001A01T01.FP_PARAM.Alarm_Hyst" : Real AT %DB5052.DBD84, 500 ms
   "2920RS001A01T01.FP_PARAM.AlarmLimit_H3" : Real AT %DB5052.DBD88, 500 ms
   "2920RS001A01T01.FP_PARAM.AlarmLimit_H2" : Real AT %DB5052.DBD92, 500 ms
   "2920RS001A01T01.FP_PARAM.AlarmLimit_H1" : Real AT %DB5052.DBD96, 500 ms
   "2920RS001A01T01.FP_PARAM.AlarmLimit_L1" : Real AT %DB5052.DBD100, 500 ms
   "2920RS001A01T01.FP_PARAM.AlarmLimit_L2" : Real AT %DB5052.DBD104, 500 ms
   "2920RS001A01T01.FP_PARAM.AlarmLimit_L3" : Real AT %DB5052.DBD108, 500 ms
   "2920RS001A01T01.FP_PARAM.AlarmDelay_H3_Pre" : Int AT %DB5052.DBW112, 500 ms
   "2920RS001A01T01.FP_PARAM.AlarmDelay_H3_Acc" : Int AT %DB5052.DBW114, 500 ms
   "2920RS001A01T01.FP_PARAM.AlarmDelay_H2_Pre" : Int AT %DB5052.DBW116, 500 ms
   "2920RS001A01T01.FP_PARAM.AlarmDelay_H2_Acc" : Int AT %DB5052.DBW118, 500 ms
   "2920RS001A01T01.FP_PARAM.AlarmDelay_H1_Pre" : Int AT %DB5052.DBW120, 500 ms
   "2920RS001A01T01.FP_PARAM.AlarmDelay_H1_Acc" : Int AT %DB5052.DBW122, 500 ms
   "2920RS001A01T01.FP_PARAM.AlarmDelay_L1_Pre" : Int AT %DB5052.DBW124, 500 ms
   "2920RS001A01T01.FP_PARAM.AlarmDelay_L1_Acc" : Int AT %DB5052.DBW126, 500 ms
   "2920RS001A01T01.FP_PARAM.AlarmDelay_L2_Pre" : Int AT %DB5052.DBW128, 500 ms
   "2920RS001A01T01.FP_PARAM.AlarmDelay_L2_Acc" : Int AT %DB5052.DBW130, 500 ms
   "2920RS001A01T01.FP_PARAM.AlarmDelay_L3_Pre" : Int AT %DB5052.DBW132, 500 ms
   "2920RS001A01T01.FP_PARAM.AlarmDelay_L3_Acc" : Int AT %DB5052.DBW134, 500 ms
   "2920RS001A01T01.FP_PARAM.OpenLoopDelay_Pre" : Int AT %DB5052.DBW136, 500 ms
   "2920RS001A01T01.FP_PARAM.OpenLoopDelay_Acc" : Int AT %DB5052.DBW138, 500 ms
   "2920RS001A01T01.FP_PARAM.OverRangeDelay_Pre" : Int AT %DB5052.DBW140, 500 ms
   "2920RS001A01T01.FP_PARAM.OverRangeDelay_Acc" : Int AT %DB5052.DBW142, 500 ms
   "2920RS001A01T01.FP_PARAM.AuxLimit_H2_Value" : Real AT %DB5052.DBD144, 500 ms
   "2920RS001A01T01.FP_PARAM.AuxLimit_H1_Value" : Real AT %DB5052.DBD148, 500 ms
   "2920RS001A01T01.FP_PARAM.AuxLimit_L2_Value" : Real AT %DB5052.DBD152, 500 ms
   "2920RS001A01T01.FP_PARAM.AuxLimit_L1_Value" : Real AT %DB5052.DBD156, 500 ms
   "2920RS001A01T01.Unit" : TextRef, internal   // Еденицы измерения При експорте из ECS через скрипт заполняется автоматически, если теги копируются в ручную то требуется задатать свойство Text
   "2920RS001A01T01.Decimals" : TextRef, internal   // Формат отображения При експорте из ECS через скрипт, заполняется автоматически. Если теги копируются в ручную то требуется задатать свойство Text s999999.9
   "2920RS001A01T01.FP_EN.Square" : Bool AT %DB5052.DBX46.0, 500 ms
   "2920RS001A01T01.FP_EN.SquareRoot" : Bool AT %DB5052.DBX46.1, 500 ms
   "2920RS001A01T01.FP_EN.ParentSupress" : Bool AT %DB5052.DBX46.2, 500 ms
   "2920RS001A01T01.FP_EN.ParentSupressUnit" : Bool AT %DB5052.DBX46.3, 500 ms
   "2920RS001A01T01.FP_EN.Force" : Bool AT %DB5052.DBX46.4, 500 ms
   "2920RS001A01T01.FP_EN.Damping" : Bool AT %DB5052.DBX46.5, 500 ms
   "2920RS001A01T01.FP_EN.Gradient_Pos" : Bool AT %DB5052.DBX46.6, 500 ms
   "2920RS001A01T01.FP_EN.Gradient_Neg" : Bool AT %DB5052.DBX46.7, 500 ms
   "2920RS001A01T01.FP_EN.Hysteresis" : Bool AT %DB5052.DBX47.0, 500 ms
   "2920RS001A01T01.FP_EN.Alarm_H3" : Bool AT %DB5052.DBX47.1, 500 ms
   "2920RS001A01T01.FP_EN.Alarm_H2" : Bool AT %DB5052.DBX47.2, 500 ms
   "2920RS001A01T01.FP_EN.Alarm_H1" : Bool AT %DB5052.DBX47.3, 500 ms
   "2920RS001A01T01.FP_EN.Alarm_L1" : Bool AT %DB5052.DBX47.4, 500 ms
   "2920RS001A01T01.FP_EN.Alarm_L2" : Bool AT %DB5052.DBX47.5, 500 ms
   "2920RS001A01T01.FP_EN.Alarm_L3" : Bool AT %DB5052.DBX47.6, 500 ms
   "2920RS001A01T01.FP_EN.AlarmDelay_H3" : Bool AT %DB5052.DBX47.7, 500 ms
   "2920RS001A01T01.FP_EN.AlarmDelay_H2" : Bool AT %DB5052.DBX48.0, 500 ms
   "2920RS001A01T01.FP_EN.AlarmDelay_H1" : Bool AT %DB5052.DBX48.1, 500 ms
   "2920RS001A01T01.FP_EN.AlarmDelay_L1" : Bool AT %DB5052.DBX48.2, 500 ms
   "2920RS001A01T01.FP_EN.AlarmDelay_L2" : Bool AT %DB5052.DBX48.3, 500 ms
   "2920RS001A01T01.FP_EN.AlarmDelay_L3" : Bool AT %DB5052.DBX48.4, 500 ms
   "2920RS001A01T01.FP_EN.ROC_Warn" : Bool AT %DB5052.DBX48.5, 500 ms
   "2920RS001A01T01.FP_EN.U_Range_Warn" : Bool AT %DB5052.DBX48.6, 500 ms
   "2920RS001A01T01.FP_EN.O_Range_Warn" : Bool AT %DB5052.DBX48.7, 500 ms
   "2920RS001A01T01.trend_tag_name" : TextRef, internal   // Еденицы измерения При експорте из ECS через скрипт - заполняется автоматически, если теги копируются в ручную то требуется задатать свойство Text - имя тега для тренда
   "2920RS001A01T01.DQ.AL_H3" : Bool AT %DB5052.DBX16.0, 500 ms
   "2920RS001A01T01.DQ.AL_H2" : Bool AT %DB5052.DBX16.1, 500 ms
   "2920RS001A01T01.DQ.AL_H1" : Bool AT %DB5052.DBX16.2, 500 ms
   "2920RS001A01T01.DQ.AL_L1" : Bool AT %DB5052.DBX16.3, 500 ms
   "2920RS001A01T01.DQ.AL_L2" : Bool AT %DB5052.DBX16.4, 500 ms
   "2920RS001A01T01.DQ.AL_L3" : Bool AT %DB5052.DBX16.5, 500 ms
   "2920RS001A01T01.DQ.SIG_OK" : Bool AT %DB5052.DBX16.6, 500 ms
   "2920RS001A01T01.DQ.LIM_H2" : Bool AT %DB5052.DBX16.7, 500 ms
   "2920RS001A01T01.DQ.LIM_H1" : Bool AT %DB5052.DBX17.0, 500 ms
   "2920RS001A01T01.DQ.LIM_L1" : Bool AT %DB5052.DBX17.1, 500 ms
   "2920RS001A01T01.DQ.LIM_L2" : Bool AT %DB5052.DBX17.2, 500 ms
   "2920RS001A01T01.DQ.GR_P" : Bool AT %DB5052.DBX17.3, 500 ms
   "2920RS001A01T01.DQ.GR_N" : Bool AT %DB5052.DBX17.4, 500 ms
   "2920RS001A01T01.I.IN" : Real AT %DB5052.DBD2, 500 ms
   "2920RS001A01T01.I.SIG_TYPE" : Int AT %DB5052.DBW0, 500 ms
   "2920RS001A01T01.I.FI_BUS" : Byte AT %DB5052.DBB6, 500 ms
   "2920RS001A01T01.DI.U_RANGE" : Bool AT %DB5052.DBX7.0, 500 ms
   "2920RS001A01T01.DI.O_RANGE" : Bool AT %DB5052.DBX7.1, 500 ms
   "2920RS001A01T01.DI.SIG_FAULT" : Bool AT %DB5052.DBX7.2, 500 ms
   "2920RS001A01T01.DI.EnConfig" : Bool AT %DB5052.DBX7.3, 500 ms
   "2920RS001A01T01.DI.AEN" : Bool AT %DB5052.DBX7.4, 500 ms
   "2920RS001A01T01.DI.AL_SUPR" : Bool AT %DB5052.DBX7.5, 500 ms
   "2920RS001A01T01.Q.PV_NORM" : Real AT %DB5052.DBD8, 500 ms
   "2920RS001A01T01.Q.PV_SCAL" : Real AT %DB5052.DBD12, 500 ms
   "2920RS001A01T01.ParentInfo" : TextRef, internal   // Имя родителя для попап окна, вкладка инфо. При експорте из ECS через скрипт заполняется автоматически, если теги копируются в ручную то требуется в ручную задатать свойство Start Value

